  MoveC 3760 to (-84.5, 214.85, -40) mm, rotated rx 180 ry 0 rz 0.01 deg; joints [38.909, -46.829, 108.857, -137.77, 69.186, 163.004] to (-86.38, 214.39, -40) mm, rotated rx 180 ry 0 rz 0.01 deg; joints [38.847, -46.78, 108.752, -137.818, 69.125, 162.986]
  MoveC 3761 to (-98.15, 202.83, -40) mm, rotated rx 180 ry 0 rz 0.01 deg; joints [38.199, -46.687, 108.571, -138.455, 68.856, 163.166] to (-111.4, 193.01, -40) mm, rotated rx -180 ry 0 rz 0.01 deg; joints [37.571, -46.495, 108.172, -139.042, 68.504, 163.259]
  MoveC 3762 to (-125.84, 185.04, -40) mm, rotated rx -180 ry 0 rz 0.01 deg; joints [36.977, -46.211, 107.571, -139.567, 68.079, 163.268] to (-141.16, 178.95, -40) mm, rotated rx -180 ry 0 rz 0.01 deg; joints [36.427, -45.844, 106.785, -140.021, 67.589, 163.195]
  MoveC 3763 to (-159.21, 174.61, -40) mm, rotated rx 180 ry 0 rz 0.01 deg; joints [35.877, -45.331, 105.687, -140.431, 66.966, 163.013] to (-177.73, 173.15, -40) mm, rotated rx 180 ry 0 rz 0.01 deg; joints [35.415, -44.722, 104.377, -140.715, 66.278, 162.723]
  MoveL 3764 to (-214.9, 173.15, -40) mm, rotated rx 180 ry 0 rz 0.01 deg; joints [34.605, -43.391, 101.519, -141.119, 64.829, 162.022]
  MoveC 3765 to (-246.16, 177.17, -40) mm, rotated rx 180 ry 0 rz 0.01 deg; joints [34.072, -42.131, 98.82, -141.24, 63.528, 161.269] to (-275.4, 188.95, -40) mm, rotated rx 180 ry 0 rz 0.01 deg; joints [33.832, -40.711, 95.78, -140.971, 62.183, 160.244]
  MoveC 3766 to (-277.77, 191.44, -40) mm, rotated rx -180 ry 0 rz 0.01 deg; joints [33.859, -40.555, 95.444, -140.883, 62.053, 160.102] to (-278.34, 194.83, -40) mm, rotated rx 180 ry 0 rz 0.01 deg; joints [33.949, -40.446, 95.207, -140.745, 61.987, 159.965]
  MoveC 3767 to (-278.82, 198.21, -40) mm, rotated rx 180 ry 0 rz 0.01 deg; joints [34.04, -40.34, 94.977, -140.606, 61.924, 159.83] to (-281, 200.83, -40) mm, rotated rx 180 ry 0 rz 0.01 deg; joints [34.075, -40.185, 94.646, -140.51, 61.8, 159.685]
  MoveC 3768 to (-299.48, 216.47, -40) mm, rotated rx 180 ry 0 rz 0.01 deg; joints [34.167, -39.034, 92.185, -139.955, 60.828, 158.683] to (-314.43, 235.5, -40) mm, rotated rx 180 ry 0 rz 0.01 deg; joints [34.423, -37.901, 89.767, -139.21, 59.951, 157.588]
  MoveC 3769 to (-316.14, 236.14, -40) mm, rotated rx -180 ry 0 rz 0.01 deg; joints [34.408, -37.812, 89.579, -139.189, 59.87, 157.521] to (-317.24, 234.68, -40) mm, rotated rx -180 ry 0 rz 0.01 deg; joints [34.344, -37.807, 89.57, -139.255, 59.841, 157.552]
  MoveL 3770 to (-317.23, 140.25, -40) mm, rotated rx -180 ry 0 rz 0.01 deg; joints [31.537, -40.248, 94.881, -143.267, 61.027, 161.125]
  MoveC 3771 to (-316.14, 136.25, -40) mm, rotated rx 180 ry 0 rz 0.01 deg; joints [31.435, -40.388, 95.185, -143.43, 61.123, 161.29] to (-313.16, 133.37, -40) mm, rotated rx -180 ry 0 rz 0.01 deg; joints [31.402, -40.577, 95.59, -143.536, 61.286, 161.455]
  MoveC 3772 to (-302.92, 127.1, -40) mm, rotated rx 180 ry 0 rz 0.01 deg; joints [31.401, -41.135, 96.786, -143.742, 61.799, 161.885] to (-293.34, 119.87, -40) mm, rotated rx 180 ry 0 rz 0.01 deg; joints [31.358, -41.682, 97.963, -143.985, 62.294, 162.328]
  MoveC 3773 to (-284.52, 111.72, -40) mm, rotated rx -180 ry 0 rz 0.01 deg; joints [31.27, -42.213, 99.11, -144.266, 62.764, 162.779] to (-276.59, 102.69, -40) mm, rotated rx 180 ry 0 rz 0.01 deg; joints [31.136, -42.723, 100.215, -144.586, 63.206, 163.234]
  MoveC 3774 to (-269.25, 92.45, -40) mm, rotated rx 180 ry 0 rz 0.01 deg; joints [30.95, -43.231, 101.321, -144.957, 63.637, 163.71] to (-262.89, 81.57, -40) mm, rotated rx -180 ry 0 rz 0.01 deg; joints [30.72, -43.709, 102.366, -145.36, 64.034, 164.181]
  MoveC 3775 to (-256.94, 70.47, -40) mm, rotated rx -180 ry 0 rz 0.01 deg; joints [30.473, -44.17, 103.376, -145.773, 64.415, 164.643] to (-250.77, 59.49, -40) mm, rotated rx -180 ry 0 rz 0.01 deg; joints [30.23, -44.63, 104.388, -146.177, 64.803, 165.098]
  MoveC 3776 to (-247.69, 56.41, -40) mm, rotated rx -180 ry 0 rz 0.01 deg; joints [30.187, -44.808, 104.778, -146.277, 64.967, 165.248] to (-243.47, 55.28, -40) mm, rotated rx -180 ry 0 rz 0.01 deg; joints [30.231, -44.987, 105.167, -146.285, 65.154, 165.356]
  MoveL 3777 to (-150.05, 55.28, -40) mm, rotated rx 180 ry 0 rz 0.01 deg; joints [32.15, -48.283, 112.334, -145.198, 68.859, 166.917]
  MoveC 3778 to (-145.86, 56.4, -40) mm, rotated rx -180 ry 0 rz 0.01 deg; joints [32.28, -48.401, 112.591, -145.094, 69.006, 166.953] to (-142.79, 59.47, -40) mm, rotated rx 180 ry 0 rz 0.01 deg; joints [32.453, -48.442, 112.674, -144.924, 69.084, 166.913]
  MoveL 3779 to (-126.05, 89.53, -40) mm, rotated rx -180 ry 0 rz 0.01 deg; joints [33.855, -48.375, 112.466, -143.442, 69.327, 166.294]
  MoveC 3780 to (-117.05, 102.8, -40) mm, rotated rx 180 ry 0 rz 0.01 deg; joints [34.51, -48.386, 112.466, -142.765, 69.488, 166.042] to (-106.26, 114.65, -40) mm, rotated rx -180 ry 0 rz 0.01 deg; joints [35.159, -48.481, 112.649, -142.117, 69.732, 165.86]
  MoveC 3781 to (-93.93, 124.89, -40) mm, rotated rx 180 ry 0 rz 0.01 deg; joints [35.794, -48.653, 113.006, -141.508, 70.048, 165.751] to (-80.35, 133.4, -40) mm, rotated rx -180 ry 0 rz 0.01 deg; joints [36.405, -48.896, 113.525, -140.945, 70.427, 165.716]
  MoveC 3782 to (-77.37, 136.23, -40) mm, rotated rx 180 ry 0 rz 0.01 deg; joints [36.572, -48.927, 113.586, -140.781, 70.496, 165.678] to (-76.28, 140.19, -40) mm, rotated rx -180 ry 0 rz 0.01 deg; joints [36.73, -48.872, 113.457, -140.604, 70.482, 165.573]
  MoveL 3783 to (-76.28, 234.68, -40) mm, rotated rx 180 ry 0 rz 0.01 deg; joints [39.722, -46.589, 108.302, -136.865, 69.215, 162.474]
  MoveC 3784 to (-77.38, 236.14, -40) mm, rotated rx -180 ry 0 rz 0.01 deg; joints [39.739, -46.517, 108.143, -136.825, 69.157, 162.404] to (-79.08, 235.49, -40) mm, rotated rx -180 ry 0 rz 0.01 deg; joints [39.676, -46.479, 108.061, -136.877, 69.105, 162.395]
  MoveC 3785 to (-106.86, 204.97, -40) mm, rotated rx 180 ry 0 rz 0.01 deg; joints [38.053, -46.35, 107.836, -138.5, 68.512, 162.939] to (-143.36, 185.73, -40) mm, rotated rx -180 ry 0 rz 0.01 deg; joints [36.588, -45.605, 106.257, -139.779, 67.418, 162.929]
  MoveC 3786 to (-160.92, 181.53, -40) mm, rotated rx -180 ry 0 rz 0.01 deg; joints [36.055, -45.105, 105.187, -140.173, 66.811, 162.749] to (-178.91, 180.18, -40) mm, rotated rx 180 ry 0 rz 0.01 deg; joints [35.608, -44.51, 103.908, -140.444, 66.141, 162.462]
  MoveL 3787 to (-214.9, 180.27, -40) mm, rotated rx 180 ry 0 rz 0.01 deg; joints [34.825, -43.217, 101.133, -140.827, 64.738, 161.775]
  MoveC 3788 to (-244.28, 184.04, -40) mm, rotated rx -180 ry 0 rz 0.01 deg; joints [34.32, -42.031, 98.596, -140.941, 63.517, 161.063] to (-271.76, 195.1, -40) mm, rotated rx -180 ry 0 rz 0.01 deg; joints [34.09, -40.696, 95.739, -140.69, 62.255, 160.095]
  MoveC 3789 to (-276.45, 197.86, -40) mm, rotated rx -180 ry 0 rz 0.01 deg; joints [34.078, -40.442, 95.195, -140.606, 62.027, 159.894] to (-281, 200.83, -40) mm, rotated rx 180 ry 0 rz 0.01 deg; joints [34.075, -40.185, 94.646, -140.51, 61.8, 159.685]
  MoveC 3790 to (-282.99, 203.32, -40) mm, rotated rx 180 ry 0 rz 0.01 deg; joints [34.109, -40.042, 94.339, -140.418, 61.686, 159.549] to (-283.24, 206.49, -40) mm, rotated rx -180 ry 0 rz 0.01 deg; joints [34.198, -39.949, 94.137, -140.287, 61.635, 159.425]
  MoveC 3791 to (-283.44, 209.65, -40) mm, rotated rx 180 ry 0 rz 0.01 deg; joints [34.287, -39.859, 93.94, -140.156, 61.587, 159.301] to (-285.27, 212.23, -40) mm, rotated rx 180 ry 0 rz 0.01 deg; joints [34.327, -39.718, 93.638, -140.058, 61.478, 159.164]
  MoveC 3792 to (-293.65, 219.64, -40) mm, rotated rx -180 ry 0 rz 0.01 deg; joints [34.376, -39.185, 92.499, -139.792, 61.034, 158.693] to (-301.3, 227.8, -40) mm, rotated rx -180 ry 0 rz 0.01 deg; joints [34.461, -38.654, 91.365, -139.485, 60.607, 158.202]
  MoveC 3793 to (-306.53, 234.56, -40) mm, rotated rx 180 ry 0 rz 0.01 deg; joints [34.553, -38.254, 90.512, -139.22, 60.3, 157.813] to (-311.05, 241.82, -40) mm, rotated rx -180 ry 0 rz 0.01 deg; joints [34.672, -37.866, 89.683, -138.929, 60.015, 157.416]
  MoveC 3794 to (-314.94, 249.42, -40) mm, rotated rx -180 ry 0 rz 0.01 deg; joints [34.812, -37.489, 88.879, -138.618, 59.751, 157.015] to (-318.34, 257.27, -40) mm, rotated rx 180 ry 0 rz 0.01 deg; joints [34.968, -37.123, 88.098, -138.292, 59.505, 156.611]
  MoveC 3795 to (-321.51, 259.02, -40) mm, rotated rx 180 ry 0 rz 0.01 deg; joints [34.955, -36.939, 87.708, -138.225, 59.346, 156.46] to (-323.82, 256.23, -40) mm, rotated rx -180 ry 0 rz 0.01 deg; joints [34.83, -36.921, 87.676, -138.351, 59.282, 156.516]
  MoveL 3796 to (-323.81, 135.87, -40) mm, rotated rx 180 ry 0 rz 0.01 deg; joints [31.279, -40.086, 94.544, -143.485, 60.797, 161.143]
  MoveC 3797 to (-322.72, 132.05, -40) mm, rotated rx -180 ry 0 rz 0.01 deg; joints [31.182, -40.222, 94.838, -143.642, 60.892, 161.302] to (-319.77, 129.39, -40) mm, rotated rx -180 ry 0 rz 0.01 deg; joints [31.155, -40.405, 95.231, -143.74, 61.051, 161.459]
  MoveC 3798 to (-299.02, 116.16, -40) mm, rotated rx -180 ry 0 rz 0.01 deg; joints [31.134, -41.544, 97.675, -144.179, 62.099, 162.343] to (-281.76, 98.61, -40) mm, rotated rx 180 ry 0 rz 0.01 deg; joints [30.907, -42.615, 99.991, -144.796, 63.041, 163.272]
  MoveC 3799 to (-273.96, 87.77, -40) mm, rotated rx 180 ry 0 rz 0.01 deg; joints [30.708, -43.154, 101.164, -145.191, 63.499, 163.776] to (-267.18, 76.25, -40) mm, rotated rx -180 ry 0 rz 0.01 deg; joints [30.465, -43.661, 102.272, -145.619, 63.921, 164.274]
  MoveL 3800 to (-254.5, 52.76, -40) mm, rotated rx 180 ry 0 rz 0.01 deg; joints [29.935, -44.63, 104.401, -146.494, 64.732, 165.243]
  MoveC 3801 to (-251.61, 49.79, -40) mm, rotated rx 180 ry 0 rz 0.01 deg; joints [29.891, -44.798, 104.77, -146.592, 64.887, 165.385] to (-247.62, 48.7, -40) mm, rotated rx -180 ry 0 rz 0.01 deg; joints [29.932, -44.969, 105.14, -146.6, 65.064, 165.488]
  MoveL 3802 to (-145.88, 48.7, -40) mm, rotated rx 180 ry 0 rz 0.01 deg; joints [32.013, -48.555, 112.946, -145.415, 69.104, 167.177]
  MoveC 3803 to (-141.9, 49.79, -40) mm, rotated rx 180 ry 0 rz 0.01 deg; joints [32.137, -48.667, 113.189, -145.314, 69.243, 167.209] to (-139.04, 52.76, -40) mm, rotated rx -180 ry 0 rz 0.01 deg; joints [32.303, -48.703, 113.262, -145.15, 69.314, 167.169]
  MoveL 3804 to (-119.94, 86.41, -40) mm, rotated rx 180 ry 0 rz 0.01 deg; joints [33.889, -48.642, 113.058, -143.48, 69.597, 166.488]
  MoveC 3805 to (-108.73, 102.26, -40) mm, rotated rx 180 ry 0 rz 0.01 deg; joints [34.685, -48.67, 113.089, -142.66, 69.805, 166.197] to (-95.08, 116.07, -40) mm, rotated rx 180 ry 0 rz 0.01 deg; joints [35.472, -48.811, 113.37, -141.885, 70.124, 166.003]
  MoveC 3806 to (-90.13, 119.96, -40) mm, rotated rx -180 ry 0 rz 0.01 deg; joints [35.72, -48.884, 113.523, -141.647, 70.253, 165.967] to (-84.87, 123.41, -40) mm, rotated rx 180 ry 0 rz 0.01 deg; joints [35.963, -48.975, 113.718, -141.422, 70.398, 165.949]
  MoveC 3807 to (-79.39, 126.51, -40) mm, rotated rx -180 ry 0 rz 0.01 deg; joints [36.199, -49.08, 113.943, -141.207, 70.554, 165.945] to (-73.78, 129.35, -40) mm, rotated rx 180 ry 0 rz 0.01 deg; joints [36.432, -49.194, 114.189, -140.999, 70.719, 165.951]
  MoveC 3808 to (-70.8, 132, -40) mm, rotated rx -180 ry 0 rz 0.01 deg; joints [36.593, -49.229, 114.259, -140.842, 70.79, 165.92] to (-69.7, 135.82, -40) mm, rotated rx 180 ry 0 rz 0.01 deg; joints [36.747, -49.178, 114.139, -140.669, 70.777, 165.82]
  MoveL 3809 to (-69.7, 256.21, -40) mm, rotated rx -180 ry 0 rz 0.01 deg; joints [40.537, -46.238, 107.505, -135.924, 69.16, 161.843]
  MoveC 3810 to (-72.01, 259, -40) mm, rotated rx -180 ry 0 rz 0.01 deg; joints [40.562, -46.091, 107.182, -135.853, 69.042, 161.703] to (-75.18, 257.25, -40) mm, rotated rx 180 ry 0 rz 0.01 deg; joints [40.429, -46.036, 107.066, -135.97, 68.954, 161.707]
  MoveC 3811 to (-85.01, 238.11, -40) mm, rotated rx -180 ry 0 rz 0.01 deg; joints [39.607, -46.221, 107.498, -136.867, 68.859, 162.198] to (-98.4, 221.27, -40) mm, rotated rx 180 ry 0 rz 0.01 deg; joints [38.762, -46.218, 107.52, -137.731, 68.602, 162.536]
  MoveC 3812 to (-114.74, 207.28, -40) mm, rotated rx 180 ry 0 rz 0.01 deg; joints [37.934, -46.033, 107.145, -138.523, 68.194, 162.718] to (-133.35, 196.51, -40) mm, rotated rx -180 ry 0 rz 0.01 deg; joints [37.158, -45.679, 106.398, -139.212, 67.65, 162.746]
  MoveC 3813 to (-152.99, 189.8, -40) mm, rotated rx 180 ry 0 rz 0.01 deg; joints [36.493, -45.176, 105.325, -139.74, 67.003, 162.615] to (-173.6, 187.26, -40) mm, rotated rx -180 ry 0 rz 0.01 deg; joints [35.946, -44.524, 103.925, -140.095, 66.254, 162.32]
  MoveL 3814 to (-214.9, 186.85, -40) mm, rotated rx -180 ry 0 rz 0.01 deg; joints [35.027, -43.054, 100.774, -140.558, 64.654, 161.546]
  MoveC 3815 to (-239.37, 189.64, -40) mm, rotated rx 180 ry 0 rz 0.01 deg; joints [34.593, -42.076, 98.682, -140.668, 63.644, 160.962] to (-262.59, 197.85, -40) mm, rotated rx 180 ry 0 rz 0.01 deg; joints [34.36, -40.982, 96.341, -140.512, 62.598, 160.188]
  MoveC 3816 to (-274.33, 204.41, -40) mm, rotated rx 180 ry 0 rz 0.01 deg; joints [34.316, -40.356, 95.001, -140.319, 62.032, 159.696] to (-285.27, 212.23, -40) mm, rotated rx 180 ry 0 rz 0.01 deg; joints [34.327, -39.718, 93.638, -140.058, 61.478, 159.164]
  MoveC 3817 to (-287.81, 216, -40) mm, rotated rx -180 ry 0 rz 0.01 deg; joints [34.386, -39.517, 93.206, -139.914, 61.325, 158.964] to (-287.78, 220.54, -40) mm, rotated rx 180 ry 0 rz 0.01 deg; joints [34.52, -39.397, 92.945, -139.724, 61.268, 158.791]
  MoveC 3818 to (-287.6, 225.04, -40) mm, rotated rx 180 ry 0 rz 0.01 deg; joints [34.656, -39.283, 92.697, -139.534, 61.218, 158.622] to (-289.76, 229, -40) mm, rotated rx 180 ry 0 rz 0.01 deg; joints [34.727, -39.089, 92.282, -139.379, 61.078, 158.421]
  MoveC 3819 to (-292.01, 231.41, -40) mm, rotated rx -180 ry 0 rz 0.01 deg; joints [34.752, -38.933, 91.949, -139.289, 60.953, 158.276] to (-294.19, 233.88, -40) mm, rotated rx 180 ry 0 rz 0.01 deg; joints [34.78, -38.777, 91.616, -139.195, 60.83, 158.129]
  MoveC 3820 to (-299.55, 240.88, -40) mm, rotated rx 180 ry 0 rz 0.01 deg; joints [34.875, -38.366, 90.738, -138.924, 60.515, 157.728] to (-304.11, 248.43, -40) mm, rotated rx 180 ry 0 rz 0.01 deg; joints [35, -37.967, 89.887, -138.623, 60.225, 157.319]
  MoveC 3821 to (-307.93, 256.38, -40) mm, rotated rx 180 ry 0 rz 0.01 deg; joints [35.15, -37.584, 89.069, -138.298, 59.961, 156.905] to (-311.05, 264.62, -40) mm, rotated rx 180 ry 0 rz 0.01 deg; joints [35.321, -37.218, 88.285, -137.957, 59.722, 156.491]
  MoveC 3822 to (-313.15, 267.5, -40) mm, rotated rx -180 ry 0 rz 0.01 deg; joints [35.36, -37.046, 87.92, -137.84, 59.595, 156.32] to (-316.54, 268.59, -40) mm, rotated rx 180 ry 0 rz 0.01 deg; joints [35.323, -36.871, 87.552, -137.802, 59.436, 156.189]
  MoveL 3823 to (-329.33, 268.59, -40) mm, rotated rx 180 ry 0 rz 0.01 deg; joints [35.07, -36.326, 86.408, -137.829, 58.884, 155.86]
  MoveC 3824 to (-332.05, 267.47, -40) mm, rotated rx 180 ry 0 rz 0.01 deg; joints [34.985, -36.242, 86.234, -137.882, 58.78, 155.837] to (-333.18, 264.74, -40) mm, rotated rx -180 ry 0 rz 0.01 deg; joints [34.886, -36.274, 86.304, -138.002, 58.766, 155.922]
  MoveL 3825 to (-333.17, 129.66, -40) mm, rotated rx 180 ry 0 rz 0.01 deg; joints [30.915, -39.85, 94.055, -143.793, 60.468, 161.167]
  MoveC 3826 to (-332.04, 125.85, -40) mm, rotated rx 180 ry 0 rz 0.01 deg; joints [30.819, -39.987, 94.352, -143.95, 60.564, 161.327] to (-329, 123.29, -40) mm, rotated rx -180 ry 0 rz 0.01 deg; joints [30.796, -40.172, 94.749, -144.045, 60.727, 161.483]
  MoveC 3827 to (-321.93, 119.98, -40) mm, rotated rx 180 ry 0 rz 0.01 deg; joints [30.824, -40.538, 95.531, -144.15, 61.074, 161.747] to (-315.03, 116.31, -40) mm, rotated rx 180 ry 0 rz 0.01 deg; joints [30.838, -40.902, 96.309, -144.269, 61.415, 162.016]
  MoveC 3828 to (-308.46, 112.08, -40) mm, rotated rx 180 ry 0 rz 0.01 deg; joints [30.828, -41.263, 97.084, -144.409, 61.748, 162.295] to (-302.39, 107.15, -40) mm, rotated rx -180 ry 0 rz 0.01 deg; joints [30.787, -41.616, 97.845, -144.58, 62.066, 162.585]
  MoveC 3829 to (-296.35, 101.27, -40) mm, rotated rx 180 ry 0 rz 0.01 deg; joints [30.715, -41.987, 98.647, -144.788, 62.394, 162.903] to (-290.71, 95, -40) mm, rotated rx 180 ry 0 rz 0.01 deg; joints [30.622, -42.348, 99.427, -145.013, 62.709, 163.222]
  MoveC 3830 to (-285.57, 88.3, -40) mm, rotated rx -180 ry 0 rz 0.01 deg; joints [30.505, -42.695, 100.182, -145.258, 63.007, 163.542] to (-281.04, 81.19, -40) mm, rotated rx -180 ry 0 rz 0.01 deg; joints [30.361, -43.025, 100.901, -145.523, 63.283, 163.86]
  MoveL 3831 to (-263.18, 49.54, -40) mm, rotated rx 180 ry 0 rz 0.01 deg; joints [29.663, -44.371, 103.849, -146.707, 64.411, 165.192]
  MoveC 3832 to (-262.37, 48.04, -40) mm, rotated rx 180 ry 0 rz 0.01 deg; joints [29.628, -44.432, 103.984, -146.763, 64.463, 165.253] to (-261.64, 46.49, -40) mm, rotated rx -180 ry 0 rz 0.01 deg; joints [29.59, -44.491, 104.114, -146.821, 64.512, 165.314]
  MoveC 3833 to (-260.94, 44.92, -40) mm, rotated rx -180 ry 0 rz 0.01 deg; joints [29.551, -44.549, 104.242, -146.881, 64.56, 165.374] to (-260.23, 43.36, -40) mm, rotated rx -180 ry 0 rz 0.01 deg; joints [29.513, -44.608, 104.37, -146.94, 64.608, 165.435]
  MoveC 3834 to (-257.69, 40.43, -40) mm, rotated rx 180 ry 0 rz 0.01 deg; joints [29.463, -44.762, 104.709, -147.041, 64.749, 165.569] to (-253.96, 39.34, -40) mm, rotated rx 180 ry 0 rz 0.01 deg; joints [29.497, -44.923, 105.059, -147.053, 64.917, 165.666]
  MoveL 3835 to (-139.55, 39.34, -40) mm, rotated rx -180 ry 0 rz 0.01 deg; joints [31.824, -48.953, 113.84, -145.717, 69.468, 167.549]
  MoveC 3836 to (-135.8, 40.44, -40) mm, rotated rx 180 ry 0 rz 0.01 deg; joints [31.944, -49.056, 114.065, -145.618, 69.597, 167.577] to (-133.25, 43.4, -40) mm, rotated rx -180 ry 0 rz 0.01 deg; joints [32.103, -49.082, 114.116, -145.458, 69.656, 167.533]
  MoveC 3837 to (-132.51, 45.06, -40) mm, rotated rx 180 ry 0 rz 0.01 deg; joints [32.178, -49.073, 114.095, -145.378, 69.663, 167.497] to (-131.77, 46.73, -40) mm, rotated rx -180 ry 0 rz 0.01 deg; joints [32.253, -49.065, 114.072, -145.298, 69.67, 167.461]
  MoveC 3838 to (-130.99, 48.39, -40) mm, rotated rx -180 ry 0 rz 0.01 deg; joints [32.328, -49.058, 114.052, -145.217, 69.678, 167.426] to (-130.12, 49.99, -40) mm, rotated rx 180 ry 0 rz 0.01 deg; joints [32.403, -49.054, 114.042, -145.138, 69.69, 167.393]
  MoveL 3839 to (-109.71, 84.93, -40) mm, rotated rx -180 ry 0 rz 0.01 deg; joints [34.074, -49.007, 113.865, -143.386, 69.999, 166.701]
  MoveC 3840 to (-97.46, 101.2, -40) mm, rotated rx 180 ry 0 rz 0.01 deg; joints [34.914, -49.057, 113.943, -142.528, 70.235, 166.416] to (-81.91, 114.34, -40) mm, rotated rx 180 ry 0 rz 0.01 deg; joints [35.73, -49.269, 114.383, -141.742, 70.627, 166.275]
  MoveC 3841 to (-77.72, 116.92, -40) mm, rotated rx 180 ry 0 rz 0.01 deg; joints [35.919, -49.345, 114.545, -141.568, 70.744, 166.266] to (-73.36, 119.19, -40) mm, rotated rx 180 ry 0 rz 0.01 deg; joints [36.102, -49.432, 114.734, -141.403, 70.871, 166.27]
  MoveC 3842 to (-68.92, 121.27, -40) mm, rotated rx 180 ry 0 rz 0.01 deg; joints [36.281, -49.526, 114.937, -141.243, 71.003, 166.28] to (-64.45, 123.31, -40) mm, rotated rx -180 ry 0 rz 0.01 deg; joints [36.46, -49.621, 115.142, -141.084, 71.135, 166.292]
  MoveC 3843 to (-61.45, 125.88, -40) mm, rotated rx 180 ry 0 rz 0.01 deg; joints [36.621, -49.657, 115.217, -140.929, 71.207, 166.263] to (-60.34, 129.67, -40) mm, rotated rx 180 ry 0 rz 0.01 deg; joints [36.775, -49.608, 115.1, -140.757, 71.196, 166.166]
  MoveL 3844 to (-60.34, 264.75, -40) mm, rotated rx 180 ry 0 rz 0.01 deg; joints [41.031, -46.308, 107.643, -135.444, 69.374, 161.712]
  MoveC 3845 to (-61.47, 267.47, -40) mm, rotated rx 180 ry 0 rz 0.01 deg; joints [41.083, -46.2, 107.404, -135.358, 69.299, 161.595] to (-64.19, 268.6, -40) mm, rotated rx 180 ry 0 rz 0.01 deg; joints [41.046, -46.083, 107.151, -135.358, 69.189, 161.506]
  MoveL 3846 to (-76.97, 268.6, -40) mm, rotated rx -180 ry 0 rz 0.01 deg; joints [40.72, -45.676, 106.271, -135.56, 68.74, 161.272]
  MoveC 3847 to (-80.36, 267.5, -40) mm, rotated rx 180 ry 0 rz 0.01 deg; joints [40.601, -45.597, 106.101, -135.654, 68.635, 161.249] to (-82.46, 264.63, -40) mm, rotated rx 180 ry 0 rz 0.01 deg; joints [40.463, -45.606, 106.125, -135.797, 68.598, 161.312]
  MoveC 3848 to (-91.11, 245.71, -40) mm, rotated rx 180 ry 0 rz 0.01 deg; joints [39.683, -45.826, 106.632, -136.664, 68.541, 161.822] to (-103.68, 229.13, -40) mm, rotated rx -180 ry 0 rz 0.01 deg; joints [38.872, -45.845, 106.701, -137.5, 68.308, 162.17]
  MoveC 3849 to (-119.33, 215.47, -40) mm, rotated rx -180 ry 0 rz 0.01 deg; joints [38.076, -45.675, 106.357, -138.264, 67.919, 162.355] to (-137.28, 205.01, -40) mm, rotated rx -180 ry 0 rz 0.01 deg; joints [37.329, -45.335, 105.642, -138.926, 67.393, 162.385]
  MoveC 3850 to (-155.98, 198.67, -40) mm, rotated rx 180 ry 0 rz 0.01 deg; joints [36.699, -44.854, 104.616, -139.421, 66.775, 162.256] to (-175.61, 196.4, -40) mm, rotated rx 180 ry 0 rz 0.01 deg; joints [36.183, -44.227, 103.271, -139.749, 66.059, 161.967]
  MoveL 3851 to (-214.9, 196.21, -40) mm, rotated rx -180 ry 0 rz 0.01 deg; joints [35.313, -42.82, 100.258, -140.175, 64.535, 161.216]
  MoveC 3852 to (-237.36, 198.78, -40) mm, rotated rx 180 ry 0 rz 0.01 deg; joints [34.912, -41.921, 98.335, -140.275, 63.608, 160.675] to (-258.67, 206.35, -40) mm, rotated rx -180 ry 0 rz 0.01 deg; joints [34.695, -40.915, 96.184, -140.13, 62.65, 159.958]
  MoveC 3853 to (-275.2, 216.32, -40) mm, rotated rx -180 ry 0 rz 0.01 deg; joints [34.651, -40.009, 94.247, -139.827, 61.844, 159.231] to (-289.76, 229, -40) mm, rotated rx -180 ry 0 rz 0.01 deg; joints [34.727, -39.089, 92.282, -139.379, 61.078, 158.421]
  MoveC 3854 to (-291.84, 233.17, -40) mm, rotated rx 180 ry 0 rz 0.01 deg; joints [34.807, -38.891, 91.858, -139.214, 60.937, 158.211] to (-291.18, 237.79, -40) mm, rotated rx -180 ry 0 rz 0.01 deg; joints [34.954, -38.792, 91.641, -139.016, 60.906, 158.045]
  MoveC 3855 to (-290.33, 242.32, -40) mm, rotated rx -180 ry 0 rz 0.01 deg; joints [35.102, -38.701, 91.443, -138.821, 60.884, 157.887] to (-291.84, 246.68, -40) mm, rotated rx 180 ry 0 rz 0.01 deg; joints [35.197, -38.519, 91.052, -138.645, 60.765, 157.68]
  MoveC 3856 to (-299.09, 259.76, -40) mm, rotated rx 180 ry 0 rz 0.01 deg; joints [35.424, -37.854, 89.63, -138.123, 60.292, 156.984] to (-303.92, 273.92, -40) mm, rotated rx 180 ry 0 rz 0.01 deg; joints [35.726, -37.245, 88.329, -137.538, 59.906, 156.286]
  MoveC 3857 to (-305.79, 276.83, -40) mm, rotated rx -180 ry 0 rz 0.01 deg; joints [35.77, -37.082, 87.981, -137.42, 59.788, 156.118] to (-309.07, 277.96, -40) mm, rotated rx 180 ry 0 rz 0.01 deg; joints [35.736, -36.911, 87.622, -137.381, 59.634, 155.989]
  MoveL 3858 to (-338.69, 277.96, -40) mm, rotated rx 180 ry 0 rz 0.01 deg; joints [35.148, -35.643, 84.962, -137.433, 58.354, 155.215]
  MoveC 3859 to (-341.41, 276.83, -40) mm, rotated rx -180 ry 0 rz 0.01 deg; joints [35.063, -35.557, 84.785, -137.484, 58.249, 155.19] to (-342.54, 274.1, -40) mm, rotated rx 180 ry 0 rz 0.01 deg; joints [34.965, -35.589, 84.856, -137.604, 58.235, 155.276]
  MoveL 3860 to (-342.54, 123.03, -40) mm, rotated rx 180 ry 0 rz 0.01 deg; joints [30.54, -39.62, 93.58, -144.116, 60.14, 161.205]
  MoveC 3861 to (-341.45, 119.5, -40) mm, rotated rx 180 ry 0 rz 0.01 deg; joints [30.451, -39.749, 93.858, -144.262, 60.231, 161.355] to (-338.56, 117.19, -40) mm, rotated rx 180 ry 0 rz 0.01 deg; joints [30.432, -39.922, 94.23, -144.348, 60.385, 161.498]
  MoveC 3862 to (-329.9, 113.43, -40) mm, rotated rx 180 ry 0 rz 0.01 deg; joints [30.474, -40.366, 95.176, -144.469, 60.808, 161.812] to (-321.53, 109.07, -40) mm, rotated rx -180 ry 0 rz 0.01 deg; joints [30.491, -40.807, 96.12, -144.611, 61.224, 162.136]
  MoveC 3863 to (-313.58, 103.96, -40) mm, rotated rx -180 ry 0 rz 0.01 deg; joints [30.478, -41.243, 97.057, -144.783, 61.628, 162.472] to (-306.25, 98, -40) mm, rotated rx 180 ry 0 rz 0.01 deg; joints [30.426, -41.67, 97.975, -144.991, 62.013, 162.821]
  MoveC 3864 to (-295.37, 86.26, -40) mm, rotated rx 180 ry 0 rz 0.01 deg; joints [30.255, -42.359, 99.466, -145.414, 62.618, 163.424] to (-286.65, 72.84, -40) mm, rotated rx -180 ry 0 rz 0.01 deg; joints [29.985, -42.989, 100.838, -145.917, 63.149, 164.029]
  MoveL 3865 to (-271.16, 44.94, -40) mm, rotated rx 180 ry 0 rz 0.01 deg; joints [29.36, -44.164, 103.412, -146.969, 64.134, 165.195]
  MoveC 3866 to (-269.8, 42.33, -40) mm, rotated rx -180 ry 0 rz 0.01 deg; joints [29.298, -44.269, 103.642, -147.067, 64.223, 165.301] to (-268.65, 39.62, -40) mm, rotated rx -180 ry 0 rz 0.01 deg; joints [29.229, -44.367, 103.859, -147.172, 64.303, 165.405]
  MoveC 3867 to (-267.59, 36.86, -40) mm, rotated rx 180 ry 0 rz 0.01 deg; joints [29.157, -44.462, 104.07, -147.279, 64.38, 165.508] to (-266.49, 34.13, -40) mm, rotated rx -180 ry 0 rz 0.01 deg; joints [29.086, -44.558, 104.282, -147.385, 64.459, 165.611]
  MoveC 3868 to (-264.02, 31.11, -40) mm, rotated rx 180 ry 0 rz 0.01 deg; joints [29.031, -44.711, 104.618, -147.49, 64.598, 165.746] to (-260.29, 29.98, -40) mm, rotated rx 180 ry 0 rz 0.01 deg; joints [29.063, -44.874, 104.971, -147.505, 64.767, 165.844]
  MoveL 3869 to (-133.15, 29.98, -40) mm, rotated rx -180 ry 0 rz 0.01 deg; joints [31.633, -49.348, 114.732, -146.018, 69.835, 167.917]
  MoveC 3870 to (-129.52, 31.07, -40) mm, rotated rx 180 ry 0 rz 0.01 deg; joints [31.751, -49.447, 114.949, -145.92, 69.959, 167.943] to (-127.1, 34, -40) mm, rotated rx 180 ry 0 rz 0.01 deg; joints [31.908, -49.47, 114.993, -145.762, 70.014, 167.899]
  MoveC 3871 to (-125.92, 36.87, -40) mm, rotated rx -180 ry 0 rz 0.01 deg; joints [32.036, -49.452, 114.949, -145.624, 70.021, 167.836] to (-124.8, 39.77, -40) mm, rotated rx 180 ry 0 rz 0.01 deg; joints [32.163, -49.432, 114.898, -145.487, 70.026, 167.772]
  MoveC 3872 to (-123.59, 42.63, -40) mm, rotated rx -180 ry 0 rz 0.01 deg; joints [32.29, -49.416, 114.855, -145.349, 70.034, 167.709] to (-122.15, 45.39, -40) mm, rotated rx 180 ry 0 rz 0.01 deg; joints [32.419, -49.408, 114.833, -145.213, 70.053, 167.653]
  MoveL 3873 to (-103.09, 78.38, -40) mm, rotated rx -180 ry 0 rz 0.01 deg; joints [34.002, -49.359, 114.654, -143.554, 70.332, 167.003]
  MoveC 3874 to (-91.51, 93.98, -40) mm, rotated rx -180 ry 0 rz 0.01 deg; joints [34.81, -49.402, 114.718, -142.729, 70.551, 166.73] to (-76.7, 106.56, -40) mm, rotated rx 180 ry 0 rz 0.01 deg; joints [35.594, -49.603, 115.136, -141.972, 70.921, 166.597]
  MoveC 3875 to (-71.53, 109.71, -40) mm, rotated rx 180 ry 0 rz 0.01 deg; joints [35.827, -49.697, 115.338, -141.756, 71.066, 166.587] to (-66.12, 112.43, -40) mm, rotated rx -180 ry 0 rz 0.01 deg; joints [36.052, -49.807, 115.576, -141.554, 71.224, 166.594]
  MoveC 3876 to (-60.57, 114.85, -40) mm, rotated rx 180 ry 0 rz 0.01 deg; joints [36.271, -49.927, 115.837, -141.36, 71.39, 166.613] to (-54.97, 117.14, -40) mm, rotated rx -180 ry 0 rz 0.01 deg; joints [36.488, -50.051, 116.105, -141.168, 71.558, 166.636]
  MoveC 3877 to (-52.07, 119.47, -40) mm, rotated rx -180 ry 0 rz 0.01 deg; joints [36.64, -50.089, 116.186, -141.023, 71.63, 166.613] to (-50.97, 123.03, -40) mm, rotated rx 180 ry 0 rz 0.01 deg; joints [36.787, -50.045, 116.08, -140.86, 71.62, 166.524]
  MoveL 3878 to (-50.98, 274.11, -40) mm, rotated rx 180 ry 0 rz 0.01 deg; joints [41.551, -46.351, 107.721, -134.932, 69.575, 161.55]
  MoveC 3879 to (-52.11, 276.84, -40) mm, rotated rx -180 ry 0 rz 0.01 deg; joints [41.601, -46.242, 107.481, -134.846, 69.499, 161.432] to (-54.83, 277.96, -40) mm, rotated rx -180 ry 0 rz 0.01 deg; joints [41.564, -46.127, 107.229, -134.848, 69.39, 161.343]
  MoveL 3880 to (-84.49, 277.96, -40) mm, rotated rx -180 ry 0 rz 0.01 deg; joints [40.804, -45.181, 105.188, -135.312, 68.351, 160.797]
  MoveC 3881 to (-87.75, 276.83, -40) mm, rotated rx 180 ry 0 rz 0.01 deg; joints [40.689, -45.106, 105.028, -135.405, 68.25, 160.777] to (-89.6, 273.92, -40) mm, rotated rx 180 ry 0 rz 0.01 deg; joints [40.557, -45.125, 105.073, -135.545, 68.222, 160.847]
  MoveC 3882 to (-96.33, 255.35, -40) mm, rotated rx -180 ry 0 rz 0.01 deg; joints [39.841, -45.403, 105.702, -136.365, 68.227, 161.386] to (-107.12, 238.8, -40) mm, rotated rx -180 ry 0 rz 0.01 deg; joints [39.08, -45.482, 105.901, -137.17, 68.056, 161.77]
  MoveC 3883 to (-121.34, 225.1, -40) mm, rotated rx 180 ry 0 rz 0.01 deg; joints [38.321, -45.363, 105.668, -137.911, 67.718, 161.985] to (-138.23, 214.88, -40) mm, rotated rx 180 ry 0 rz 0.01 deg; joints [37.609, -45.055, 105.019, -138.545, 67.229, 162.027]
  MoveC 3884 to (-147.91, 210.98, -40) mm, rotated rx -180 ry 0 rz 0.01 deg; joints [37.263, -44.823, 104.528, -138.826, 66.919, 161.982] to (-157.92, 208.04, -40) mm, rotated rx 180 ry 0 rz 0.01 deg; joints [36.942, -44.553, 103.951, -139.069, 66.581, 161.897]
  MoveC 3885 to (-168.2, 206.2, -40) mm, rotated rx 180 ry 0 rz 0.01 deg; joints [36.651, -44.242, 103.286, -139.268, 66.215, 161.767] to (-178.62, 205.58, -40) mm, rotated rx -180 ry 0 rz 0.01 deg; joints [36.396, -43.891, 102.534, -139.413, 65.825, 161.59]
  MoveL 3886 to (-217.25, 205.68, -40) mm, rotated rx -180 ry 0 rz 0.01 deg; joints [35.549, -42.494, 99.545, -139.811, 64.321, 160.832]
  MoveC 3887 to (-236.55, 208.01, -40) mm, rotated rx -180 ry 0 rz 0.01 deg; joints [35.207, -41.715, 97.882, -139.888, 63.523, 160.357] to (-254.82, 214.67, -40) mm, rotated rx -180 ry 0 rz 0.01 deg; joints [35.022, -40.846, 96.025, -139.758, 62.701, 159.732]
  MoveC 3888 to (-271.56, 225.24, -40) mm, rotated rx 180 ry 0 rz 0.01 deg; joints [34.988, -39.915, 94.034, -139.433, 61.881, 158.973] to (-285.89, 238.89, -40) mm, rotated rx 180 ry 0 rz 0.01 deg; joints [35.093, -38.975, 92.025, -138.943, 61.113, 158.124]
  MoveC 3889 to (-288.98, 242.7, -40) mm, rotated rx 180 ry 0 rz 0.01 deg; joints [35.14, -38.745, 91.535, -138.799, 60.936, 157.904] to (-291.84, 246.68, -40) mm, rotated rx 180 ry 0 rz 0.01 deg; joints [35.197, -38.519, 91.052, -138.645, 60.765, 157.68]
  MoveC 3890 to (-293.12, 250.97, -40) mm, rotated rx -180 ry 0 rz 0.01 deg; joints [35.294, -38.347, 90.682, -138.47, 60.656, 157.48] to (-291.71, 255.22, -40) mm, rotated rx -180 ry 0 rz 0.01 deg; joints [35.444, -38.285, 90.545, -138.284, 60.661, 157.343]
  MoveC 3891 to (-290.12, 259.34, -40) mm, rotated rx 180 ry 0 rz 0.01 deg; joints [35.594, -38.233, 90.429, -138.103, 60.675, 157.216] to (-290.76, 263.71, -40) mm, rotated rx 180 ry 0 rz 0.01 deg; joints [35.705, -38.083, 90.106, -137.922, 60.592, 157.025]
  MoveC 3892 to (-291.59, 265.76, -40) mm, rotated rx -180 ry 0 rz 0.01 deg; joints [35.746, -37.99, 89.907, -137.839, 60.53, 156.922] to (-292.37, 267.83, -40) mm, rotated rx 180 ry 0 rz 0.01 deg; joints [35.789, -37.899, 89.712, -137.754, 60.471, 156.819]
  MoveC 3893 to (-294.26, 273.68, -40) mm, rotated rx -180 ry 0 rz 0.01 deg; joints [35.916, -37.652, 89.184, -137.514, 60.316, 156.534] to (-295.79, 279.64, -40) mm, rotated rx -180 ry 0 rz 0.01 deg; joints [36.052, -37.415, 88.677, -137.267, 60.175, 156.251]
  MoveC 3894 to (-295.98, 280.55, -40) mm, rotated rx 180 ry 0 rz 0.01 deg; joints [36.074, -37.38, 88.603, -137.229, 60.155, 156.209] to (-296.14, 281.47, -40) mm, rotated rx -180 ry 0 rz 0.01 deg; joints [36.096, -37.347, 88.531, -137.191, 60.137, 156.167]
  MoveC 3895 to (-296.3, 282.38, -40) mm, rotated rx 180 ry 0 rz 0.01 deg; joints [36.119, -37.313, 88.46, -137.153, 60.118, 156.126] to (-296.48, 283.29, -40) mm, rotated rx 180 ry 0 rz 0.01 deg; joints [36.14, -37.279, 88.386, -137.115, 60.099, 156.083]
  MoveC 3896 to (-298.29, 286.19, -40) mm, rotated rx -180 ry 0 rz 0.01 deg; joints [36.184, -37.118, 88.044, -136.998, 59.985, 155.917] to (-301.51, 287.32, -40) mm, rotated rx -180 ry 0 rz 0.01 deg; joints [36.15, -36.95, 87.69, -136.96, 59.834, 155.789]
  MoveL 3897 to (-348.05, 287.32, -40) mm, rotated rx -180 ry 0 rz 0.01 deg; joints [35.224, -34.946, 83.49, -137.025, 57.82, 154.551]
  MoveC 3898 to (-350.78, 286.19, -40) mm, rotated rx 180 ry 0 rz 0.01 deg; joints [35.14, -34.859, 83.31, -137.074, 57.714, 154.525] to (-351.9, 283.47, -40) mm, rotated rx 180 ry 0 rz 0.01 deg; joints [35.043, -34.892, 83.383, -137.193, 57.699, 154.613]
  MoveL 3899 to (-351.9, 115.53, -40) mm, rotated rx 180 ry 0 rz 0.01 deg; joints [30.141, -39.406, 93.14, -144.473, 59.819, 161.274]
  MoveC 3900 to (-350.81, 112.32, -40) mm, rotated rx 180 ry 0 rz 0.01 deg; joints [30.061, -39.527, 93.401, -144.606, 59.906, 161.412] to (-348, 110.45, -40) mm, rotated rx 180 ry 0 rz 0.01 deg; joints [30.054, -39.688, 93.745, -144.675, 60.053, 161.539]
  MoveC 3901 to (-321.73, 98.25, -40) mm, rotated rx -180 ry 0 rz 0.01 deg; joints [30.148, -41.045, 96.645, -145.071, 61.346, 162.506] to (-301.24, 77.78, -40) mm, rotated rx 180 ry 0 rz 0.01 deg; joints [29.874, -42.313, 99.384, -145.812, 62.471, 163.594]
  MoveC 3902 to (-286.18, 53.51, -40) mm, rotated rx 180 ry 0 rz 0.01 deg; joints [29.364, -43.414, 101.785, -146.728, 63.401, 164.659] to (-273.87, 27.74, -40) mm, rotated rx -180 ry 0 rz 0.01 deg; joints [28.735, -44.407, 103.969, -147.718, 64.227, 165.681]
  MoveC 3903 to (-273.57, 26.95, -40) mm, rotated rx -180 ry 0 rz 0.01 deg; joints [28.714, -44.434, 104.028, -147.748, 64.249, 165.71] to (-273.3, 26.15, -40) mm, rotated rx 180 ry 0 rz 0.01 deg; joints [28.693, -44.46, 104.086, -147.78, 64.27, 165.739]
  MoveC 3904 to (-273.05, 25.35, -40) mm, rotated rx -180 ry 0 rz 0.01 deg; joints [28.67, -44.485, 104.142, -147.812, 64.29, 165.768] to (-272.79, 24.55, -40) mm, rotated rx 180 ry 0 rz 0.01 deg; joints [28.648, -44.511, 104.199, -147.843, 64.311, 165.797]
  MoveC 3905 to (-270.66, 21.7, -40) mm, rotated rx 180 ry 0 rz 0.01 deg; joints [28.591, -44.647, 104.499, -147.946, 64.433, 165.92] to (-267.28, 20.62, -40) mm, rotated rx -180 ry 0 rz 0.01 deg; joints [28.617, -44.796, 104.822, -147.962, 64.588, 166.01]
  MoveL 3906 to (-126.31, 20.62, -40) mm, rotated rx 180 ry 0 rz 0.01 deg; joints [31.449, -49.754, 115.651, -146.312, 70.218, 168.287]
  MoveC 3907 to (-122.89, 21.7, -40) mm, rotated rx -180 ry 0 rz 0.01 deg; joints [31.563, -49.845, 115.851, -146.216, 70.334, 168.311] to (-120.72, 24.55, -40) mm, rotated rx 180 ry 0 rz 0.01 deg; joints [31.713, -49.862, 115.881, -146.064, 70.38, 168.265]
  MoveC 3908 to (-115.57, 37.15, -40) mm, rotated rx -180 ry 0 rz 0.01 deg; joints [32.276, -49.786, 115.686, -145.458, 70.41, 167.992] to (-109.29, 49.24, -40) mm, rotated rx 180 ry 0 rz 0.01 deg; joints [32.844, -49.751, 115.583, -144.858, 70.487, 167.749]
  MoveL 3909 to (-96.03, 72.18, -40) mm, rotated rx 180 ry 0 rz 0.01 deg; joints [33.952, -49.714, 115.452, -143.698, 70.676, 167.299]
  MoveC 3910 to (-86.53, 85.34, -40) mm, rotated rx -180 ry 0 rz 0.01 deg; joints [34.632, -49.744, 115.49, -143.002, 70.85, 167.068] to (-74.56, 96.31, -40) mm, rotated rx -180 ry 0 rz 0.01 deg; joints [35.296, -49.89, 115.792, -142.354, 71.138, 166.938]
  MoveC 3911 to (-60.7, 104.74, -40) mm, rotated rx -180 ry 0 rz 0.01 deg; joints [35.924, -50.143, 116.334, -141.772, 71.523, 166.914] to (-45.52, 110.45, -40) mm, rotated rx 180 ry 0 rz 0.01 deg; joints [36.499, -50.487, 117.087, -141.27, 71.986, 166.992]
  MoveC 3912 to (-42.7, 112.35, -40) mm, rotated rx 180 ry 0 rz 0.01 deg; joints [36.635, -50.532, 117.183, -141.142, 72.06, 166.982] to (-41.61, 115.57, -40) mm, rotated rx -180 ry 0 rz 0.01 deg; joints [36.772, -50.495, 117.095, -140.992, 72.054, 166.903]
  MoveL 3913 to (-41.61, 283.47, -40) mm, rotated rx -180 ry 0 rz 0.01 deg; joints [42.071, -46.389, 107.788, -134.418, 69.772, 161.385]
  MoveC 3914 to (-42.74, 286.2, -40) mm, rotated rx 180 ry 0 rz 0.01 deg; joints [42.121, -46.28, 107.547, -134.333, 69.697, 161.267] to (-45.47, 287.33, -40) mm, rotated rx -180 ry 0 rz 0.01 deg; joints [42.082, -46.165, 107.296, -134.336, 69.589, 161.177]
  MoveL 3915 to (-91.94, 287.33, -40) mm, rotated rx -180 ry 0 rz 0.01 deg; joints [40.889, -44.683, 104.1, -135.06, 67.963, 160.316]
  MoveC 3916 to (-95.17, 286.2, -40) mm, rotated rx -180 ry 0 rz 0.01 deg; joints [40.776, -44.608, 103.941, -135.15, 67.862, 160.296] to (-97, 283.32, -40) mm, rotated rx 180 ry 0 rz 0.01 deg; joints [40.647, -44.627, 103.986, -135.288, 67.835, 160.367]
  MoveL 3917 to (-99.67, 271.84, -40) mm, rotated rx 180 ry 0 rz 0.01 deg; joints [40.245, -44.852, 104.488, -135.772, 67.89, 160.733]
  MoveC 3918 to (-101.39, 266.18, -40) mm, rotated rx 180 ry 0 rz 0.01 deg; joints [40.036, -44.948, 104.704, -136.017, 67.902, 160.905] to (-103.89, 260.82, -40) mm, rotated rx 180 ry 0 rz 0.01 deg; joints [39.817, -45.009, 104.845, -136.261, 67.883, 161.051]
  MoveC 3919 to (-117.37, 242.31, -40) mm, rotated rx -180 ry 0 rz 0.01 deg; joints [38.936, -45.051, 104.966, -137.177, 67.638, 161.457] to (-134.99, 227.68, -40) mm, rotated rx -180 ry 0 rz 0.01 deg; joints [38.074, -44.838, 104.531, -137.993, 67.182, 161.642]
  MoveC 3920 to (-155.89, 218.19, -40) mm, rotated rx -180 ry 0 rz 0.01 deg; joints [37.298, -44.366, 103.531, -138.638, 66.525, 161.581] to (-178.62, 214.94, -40) mm, rotated rx -180 ry 0 rz 0.01 deg; joints [36.681, -43.653, 102.009, -139.036, 65.704, 161.261]
  MoveL 3921 to (-221.2, 215.57, -40) mm, rotated rx -180 ry 0 rz 0.01 deg; joints [35.761, -42.094, 98.676, -139.444, 64.038, 160.396]
  MoveC 3922 to (-242.39, 219.41, -40) mm, rotated rx 180 ry 0 rz 0.01 deg; joints [35.423, -41.198, 96.764, -139.467, 63.144, 159.818] to (-261.5, 229.33, -40) mm, rotated rx 180 ry 0 rz 0.01 deg; joints [35.316, -40.2, 94.63, -139.197, 62.242, 159.038]
  MoveC 3923 to (-268.93, 235.17, -40) mm, rotated rx 180 ry 0 rz 0.01 deg; joints [35.333, -39.751, 93.671, -139.002, 61.863, 158.652] to (-275.9, 241.56, -40) mm, rotated rx -180 ry 0 rz 0.01 deg; joints [35.374, -39.301, 92.71, -138.777, 61.494, 158.249]
  MoveC 3924 to (-282.14, 248.68, -40) mm, rotated rx -180 ry 0 rz 0.01 deg; joints [35.452, -38.855, 91.757, -138.513, 61.144, 157.827] to (-287.3, 256.62, -40) mm, rotated rx -180 ry 0 rz 0.01 deg; joints [35.574, -38.424, 90.836, -138.205, 60.827, 157.392]
  MoveC 3925 to (-289.12, 260.12, -40) mm, rotated rx 180 ry 0 rz 0.01 deg; joints [35.637, -38.251, 90.467, -138.066, 60.706, 157.208] to (-290.76, 263.71, -40) mm, rotated rx 180 ry 0 rz 0.01 deg; joints [35.705, -38.083, 90.106, -137.922, 60.592, 157.025]
  MoveC 3926 to (-291.22, 268.09, -40) mm, rotated rx 180 ry 0 rz 0.01 deg; joints [35.82, -37.938, 89.795, -137.738, 60.516, 156.836] to (-289.15, 271.99, -40) mm, rotated rx 180 ry 0 rz 0.01 deg; joints [35.973, -37.91, 89.73, -137.565, 60.552, 156.728]
  MoveC 3927 to (-286.92, 275.73, -40) mm, rotated rx -180 ry 0 rz 0.01 deg; joints [36.124, -37.893, 89.688, -137.398, 60.597, 156.63] to (-286.73, 280.07, -40) mm, rotated rx 180 ry 0 rz 0.01 deg; joints [36.25, -37.774, 89.432, -137.214, 60.549, 156.456]
  MoveC 3928 to (-287.89, 286.46, -40) mm, rotated rx -180 ry 0 rz 0.01 deg; joints [36.405, -37.539, 88.929, -136.949, 60.418, 156.165] to (-288.76, 292.89, -40) mm, rotated rx 180 ry 0 rz 0.01 deg; joints [36.567, -37.313, 88.444, -136.68, 60.299, 155.877]
  MoveC 3929 to (-290.15, 295.6, -40) mm, rotated rx -180 ry 0 rz 0.01 deg; joints [36.613, -37.175, 88.149, -136.571, 60.205, 155.729] to (-293, 296.68, -40) mm, rotated rx 180 ry 0 rz 0.01 deg; joints [36.585, -37.025, 87.832, -136.534, 60.072, 155.611]
  MoveL 3930 to (-357.41, 296.68, -40) mm, rotated rx -180 ry 0 rz 0.01 deg; joints [35.299, -34.236, 81.993, -136.603, 57.28, 153.87]
  MoveC 3931 to (-360.14, 295.55, -40) mm, rotated rx 180 ry 0 rz 0.01 deg; joints [35.216, -34.147, 81.81, -136.65, 57.173, 153.841] to (-361.27, 292.83, -40) mm, rotated rx -180 ry 0 rz 0.01 deg; joints [35.12, -34.181, 81.885, -136.769, 57.158, 153.931]
  MoveL 3932 to (-361.26, 107.57, -40) mm, rotated rx 180 ry 0 rz 0.01 deg; joints [29.729, -39.198, 92.714, -144.846, 59.5, 161.358]
  MoveC 3933 to (-360.16, 104.51, -40) mm, rotated rx -180 ry 0 rz 0.01 deg; joints [29.654, -39.316, 92.967, -144.974, 59.585, 161.491] to (-357.38, 102.86, -40) mm, rotated rx -180 ry 0 rz 0.01 deg; joints [29.652, -39.471, 93.299, -145.036, 59.73, 161.61]
  MoveC 3934 to (-353.91, 102.2, -40) mm, rotated rx 180 ry 0 rz 0.01 deg; joints [29.693, -39.632, 93.641, -145.051, 59.891, 161.707] to (-350.43, 101.57, -40) mm, rotated rx -180 ry 0 rz 0.01 deg; joints [29.735, -39.792, 93.98, -145.065, 60.053, 161.802]
  MoveC 3935 to (-346.99, 100.74, -40) mm, rotated rx -180 ry 0 rz 0.01 deg; joints [29.77, -39.954, 94.325, -145.087, 60.214, 161.904] to (-343.67, 99.52, -40) mm, rotated rx -180 ry 0 rz 0.01 deg; joints [29.792, -40.12, 94.678, -145.125, 60.375, 162.015]
  MoveC 3936 to (-332.37, 93.68, -40) mm, rotated rx -180 ry 0 rz 0.01 deg; joints [29.812, -40.716, 95.955, -145.321, 60.94, 162.449] to (-321.93, 86.42, -40) mm, rotated rx 180 ry 0 rz 0.01 deg; joints [29.771, -41.301, 97.212, -145.575, 61.481, 162.906]
  MoveC 3937 to (-312.75, 77.57, -40) mm, rotated rx -180 ry 0 rz 0.01 deg; joints [29.656, -41.863, 98.424, -145.896, 61.982, 163.382] to (-305.37, 67.16, -40) mm, rotated rx -180 ry 0 rz 0.01 deg; joints [29.456, -42.379, 99.545, -146.289, 62.423, 163.865]
  MoveL 3938 to (-290.63, 42.14, -40) mm, rotated rx -180 ry 0 rz 0.01 deg; joints [28.908, -43.476, 101.94, -147.242, 63.349, 164.94]
  MoveC 3939 to (-284.15, 29.09, -40) mm, rotated rx -180 ry 0 rz 0.01 deg; joints [28.593, -43.989, 103.066, -147.744, 63.779, 165.461] to (-279.86, 15.16, -40) mm, rotated rx -180 ry 0 rz 0.01 deg; joints [28.203, -44.427, 104.036, -148.299, 64.125, 165.962]
  MoveC 3940 to (-278.11, 12.35, -40) mm, rotated rx 180 ry 0 rz 0.01 deg; joints [28.14, -44.548, 104.302, -148.404, 64.231, 166.077] to (-274.98, 11.25, -40) mm, rotated rx -180 ry 0 rz 0.01 deg; joints [28.159, -44.687, 104.605, -148.424, 64.376, 166.163]
  MoveL 3941 to (-118.59, 11.25, -40) mm, rotated rx -180 ry 0 rz 0.01 deg; joints [31.282, -50.184, 116.625, -146.593, 70.635, 168.667]
  MoveC 3942 to (-115.4, 12.38, -40) mm, rotated rx 180 ry 0 rz 0.01 deg; joints [31.393, -50.267, 116.807, -146.497, 70.741, 168.685] to (-113.62, 15.27, -40) mm, rotated rx -180 ry 0 rz 0.01 deg; joints [31.536, -50.27, 116.807, -146.348, 70.771, 168.633]
  MoveC 3943 to (-112.31, 20.67, -40) mm, rotated rx 180 ry 0 rz 0.01 deg; joints [31.76, -50.21, 116.663, -146.1, 70.75, 168.505] to (-110.67, 25.98, -40) mm, rotated rx -180 ry 0 rz 0.01 deg; joints [31.987, -50.161, 116.543, -145.852, 70.742, 168.383]
  MoveC 3944 to (-108.62, 31.15, -40) mm, rotated rx -180 ry 0 rz 0.01 deg; joints [32.218, -50.128, 116.458, -145.603, 70.751, 168.271] to (-106.07, 36.1, -40) mm, rotated rx 180 ry 0 rz 0.01 deg; joints [32.452, -50.114, 116.417, -145.357, 70.782, 168.172]
  MoveL 3945 to (-84.46, 72.66, -40) mm, rotated rx 180 ry 0 rz 0.01 deg; joints [34.241, -50.073, 116.246, -143.491, 71.096, 167.472]
  MoveC 3946 to (-75.24, 82.93, -40) mm, rotated rx 180 ry 0 rz 0.01 deg; joints [34.819, -50.151, 116.398, -142.914, 71.295, 167.322] to (-64.59, 91.72, -40) mm, rotated rx -180 ry 0 rz 0.01 deg; joints [35.381, -50.299, 116.709, -142.372, 71.561, 167.237]
  MoveC 3947 to (-52.48, 98.44, -40) mm, rotated rx 180 ry 0 rz 0.01 deg; joints [35.912, -50.531, 117.211, -141.884, 71.904, 167.236] to (-39.21, 102.39, -40) mm, rotated rx 180 ry 0 rz 0.01 deg; joints [36.382, -50.853, 117.919, -141.483, 72.321, 167.335]
  MoveC 3948 to (-38.46, 102.52, -40) mm, rotated rx 180 ry 0 rz 0.01 deg; joints [36.405, -50.873, 117.963, -141.464, 72.346, 167.344] to (-37.71, 102.62, -40) mm, rotated rx 180 ry 0 rz 0.01 deg; joints [36.428, -50.894, 118.009, -141.446, 72.371, 167.353]
  MoveC 3949 to (-36.96, 102.72, -40) mm, rotated rx -180 ry 0 rz 0.01 deg; joints [36.45, -50.914, 118.054, -141.428, 72.396, 167.362] to (-36.22, 102.84, -40) mm, rotated rx -180 ry 0 rz 0.01 deg; joints [36.473, -50.934, 118.099, -141.409, 72.421, 167.371]
  MoveC 3950 to (-33.37, 104.5, -40) mm, rotated rx 180 ry 0 rz 0.01 deg; joints [36.603, -50.985, 118.208, -141.289, 72.498, 167.368] to (-32.25, 107.6, -40) mm, rotated rx -180 ry 0 rz 0.01 deg; joints [36.738, -50.952, 118.128, -141.142, 72.494, 167.294]
  MoveL 3951 to (-32.25, 292.84, -40) mm, rotated rx -180 ry 0 rz 0.01 deg; joints [42.591, -46.422, 107.844, -133.903, 69.967, 161.218]
  MoveC 3952 to (-33.38, 295.56, -40) mm, rotated rx -180 ry 0 rz 0.01 deg; joints [42.64, -46.312, 107.603, -133.82, 69.893, 161.1] to (-36.11, 296.69, -40) mm, rotated rx -180 ry 0 rz 0.01 deg; joints [42.6, -46.198, 107.352, -133.824, 69.785, 161.009]
  MoveL 3953 to (-100.55, 296.69, -40) mm, rotated rx 180 ry 0 rz 0.01 deg; joints [40.944, -44.14, 102.92, -134.82, 67.532, 159.807]
  MoveC 3954 to (-103.38, 295.6, -40) mm, rotated rx -180 ry 0 rz 0.01 deg; joints [40.842, -44.077, 102.786, -134.902, 67.445, 159.793] to (-104.75, 292.9, -40) mm, rotated rx -180 ry 0 rz 0.01 deg; joints [40.731, -44.107, 102.854, -135.026, 67.431, 159.867]
  MoveC 3955 to (-106.47, 282.43, -40) mm, rotated rx 180 ry 0 rz 0.01 deg; joints [40.386, -44.339, 103.368, -135.456, 67.506, 160.219] to (-109.43, 272.25, -40) mm, rotated rx -180 ry 0 rz 0.01 deg; joints [40.017, -44.518, 103.77, -135.893, 67.533, 160.534]
  MoveC 3956 to (-113.76, 262.56, -40) mm, rotated rx -180 ry 0 rz 0.01 deg; joints [39.626, -44.636, 104.038, -136.332, 67.503, 160.802] to (-119.5, 253.63, -40) mm, rotated rx 180 ry 0 rz 0.01 deg; joints [39.222, -44.682, 104.152, -136.761, 67.411, 161.014]
  MoveC 3957 to (-125.72, 246.48, -40) mm, rotated rx 180 ry 0 rz 0.01 deg; joints [38.86, -44.662, 104.121, -137.126, 67.277, 161.152] to (-132.85, 240.25, -40) mm, rotated rx 180 ry 0 rz 0.01 deg; joints [38.503, -44.584, 103.965, -137.467, 67.096, 161.239]
  MoveC 3958 to (-140.69, 234.94, -40) mm, rotated rx -180 ry 0 rz 0.01 deg; joints [38.158, -44.456, 103.699, -137.779, 66.876, 161.279] to (-149.05, 230.51, -40) mm, rotated rx -180 ry 0 rz 0.01 deg; joints [37.829, -44.285, 103.337, -138.061, 66.622, 161.277]
  MoveC 3959 to (-154.63, 228.32, -40) mm, rotated rx -180 ry 0 rz 0.01 deg; joints [37.633, -44.149, 103.049, -138.217, 66.441, 161.248] to (-160.42, 226.78, -40) mm, rotated rx 180 ry 0 rz 0.01 deg; joints [37.452, -43.988, 102.706, -138.349, 66.243, 161.192]
  MoveC 3960 to (-166.3, 225.67, -40) mm, rotated rx 180 ry 0 rz 0.01 deg; joints [37.284, -43.811, 102.329, -138.463, 66.035, 161.118] to (-172.22, 224.75, -40) mm, rotated rx -180 ry 0 rz 0.01 deg; joints [37.121, -43.627, 101.937, -138.569, 65.822, 161.037]
  MoveL 3961 to (-214.9, 224.3, -40) mm, rotated rx -180 ry 0 rz 0.01 deg; joints [36.158, -42.1, 98.674, -139.029, 64.175, 160.206]
  MoveC 3962 to (-235.16, 227.22, -40) mm, rotated rx -180 ry 0 rz 0.01 deg; joints [35.808, -41.266, 96.896, -139.087, 63.334, 159.681] to (-253.77, 235.75, -40) mm, rotated rx -180 ry 0 rz 0.01 deg; joints [35.665, -40.327, 94.89, -138.878, 62.475, 158.963]
  MoveC 3963 to (-269.43, 248.83, -40) mm, rotated rx 180 ry 0 rz 0.01 deg; joints [35.718, -39.357, 92.817, -138.436, 61.668, 158.112] to (-281.43, 265.35, -40) mm, rotated rx 180 ry 0 rz 0.01 deg; joints [35.943, -38.414, 90.802, -137.81, 60.96, 157.181]
  MoveC 3964 to (-284.44, 271.87, -40) mm, rotated rx 180 ry 0 rz 0.01 deg; joints [36.066, -38.106, 90.142, -137.55, 60.751, 156.847] to (-286.46, 278.76, -40) mm, rotated rx -180 ry 0 rz 0.01 deg; joints [36.219, -37.824, 89.539, -137.268, 60.578, 156.517]
  MoveC 3965 to (-286.6, 279.42, -40) mm, rotated rx 180 ry 0 rz 0.01 deg; joints [36.235, -37.799, 89.485, -137.241, 60.564, 156.487] to (-286.73, 280.07, -40) mm, rotated rx 180 ry 0 rz 0.01 deg; joints [36.25, -37.774, 89.432, -137.214, 60.549, 156.456]
  MoveC 3966 to (-286.32, 284.45, -40) mm, rotated rx -180 ry 0 rz 0.01 deg; joints [36.381, -37.663, 89.191, -137.028, 60.51, 156.287] to (-283.54, 287.85, -40) mm, rotated rx 180 ry 0 rz 0.01 deg; joints [36.534, -37.676, 89.215, -136.873, 60.582, 156.215]
  MoveC 3967 to (-280.65, 291.08, -40) mm, rotated rx -180 ry 0 rz 0.01 deg; joints [36.684, -37.699, 89.257, -136.724, 60.66, 156.152] to (-279.67, 295.3, -40) mm, rotated rx -180 ry 0 rz 0.01 deg; joints [36.822, -37.613, 89.071, -136.542, 60.646, 156.001]
  MoveC 3968 to (-279.65, 298.86, -40) mm, rotated rx 180 ry 0 rz 0.01 deg; joints [36.922, -37.508, 88.844, -136.392, 60.601, 155.854] to (-279.43, 302.41, -40) mm, rotated rx 180 ry 0 rz 0.01 deg; joints [37.025, -37.411, 88.635, -136.242, 60.564, 155.711]
  MoveC 3969 to (-280.29, 304.96, -40) mm, rotated rx 180 ry 0 rz 0.01 deg; joints [37.077, -37.299, 88.396, -136.138, 60.496, 155.583] to (-282.75, 306.05, -40) mm, rotated rx 180 ry 0 rz 0.01 deg; joints [37.056, -37.165, 88.114, -136.101, 60.379, 155.476]
  MoveL 3970 to (-366.78, 306.04, -40) mm, rotated rx -180 ry 0 rz 0.01 deg; joints [35.373, -33.511, 80.467, -136.167, 56.735, 153.168]
  MoveC 3971 to (-369.5, 304.92, -40) mm, rotated rx 180 ry 0 rz 0.01 deg; joints [35.29, -33.421, 80.282, -136.21, 56.626, 153.137] to (-370.63, 302.19, -40) mm, rotated rx -180 ry 0 rz 0.01 deg; joints [35.195, -33.456, 80.358, -136.33, 56.611, 153.228]
  MoveL 3972 to (-370.62, 98.54, -40) mm, rotated rx 180 ry 0 rz 0.01 deg; joints [29.287, -39.01, 92.331, -145.264, 59.189, 161.48]
  MoveC 3973 to (-369.54, 95.83, -40) mm, rotated rx -180 ry 0 rz 0.01 deg; joints [29.222, -39.118, 92.564, -145.377, 59.27, 161.6] to (-366.9, 94.62, -40) mm, rotated rx 180 ry 0 rz 0.01 deg; joints [29.23, -39.259, 92.863, -145.422, 59.404, 161.7]
  MoveC 3974 to (-344.51, 89.56, -40) mm, rotated rx 180 ry 0 rz 0.01 deg; joints [29.465, -40.311, 95.101, -145.555, 60.458, 162.346] to (-325.15, 77.22, -40) mm, rotated rx 180 ry 0 rz 0.01 deg; joints [29.421, -41.374, 97.382, -145.983, 61.451, 163.153]
  MoveC 3975 to (-322.59, 74.68, -40) mm, rotated rx -180 ry 0 rz 0.01 deg; joints [29.385, -41.532, 97.724, -146.077, 61.593, 163.288] to (-320.27, 71.92, -40) mm, rotated rx 180 ry 0 rz 0.01 deg; joints [29.339, -41.685, 98.055, -146.18, 61.726, 163.425]
  MoveC 3976 to (-318.09, 69.06, -40) mm, rotated rx -180 ry 0 rz 0.01 deg; joints [29.287, -41.834, 98.378, -146.289, 61.855, 163.562] to (-315.92, 66.18, -40) mm, rotated rx -180 ry 0 rz 0.01 deg; joints [29.233, -41.982, 98.699, -146.398, 61.982, 163.699]
  MoveL 3977 to (-295.35, 31.01, -40) mm, rotated rx 180 ry 0 rz 0.01 deg; joints [28.454, -43.519, 102.053, -147.749, 63.281, 165.205]
  MoveC 3978 to (-292.39, 25.06, -40) mm, rotated rx -180 ry 0 rz 0.01 deg; joints [28.309, -43.752, 102.565, -147.979, 63.477, 165.443] to (-290.18, 18.79, -40) mm, rotated rx -180 ry 0 rz 0.01 deg; joints [28.139, -43.961, 103.026, -148.228, 63.645, 165.675]
  MoveC 3979 to (-288.66, 12.32, -40) mm, rotated rx -180 ry 0 rz 0.01 deg; joints [27.949, -44.146, 103.436, -148.49, 63.786, 165.899] to (-287.73, 5.74, -40) mm, rotated rx 180 ry 0 rz 0.01 deg; joints [27.744, -44.308, 103.799, -148.762, 63.902, 166.114]
  MoveC 3980 to (-286.36, 3, -40) mm, rotated rx -180 ry 0 rz 0.01 deg; joints [27.675, -44.413, 104.03, -148.867, 63.992, 166.22] to (-283.5, 1.89, -40) mm, rotated rx 180 ry 0 rz 0.01 deg; joints [27.689, -44.543, 104.313, -148.892, 64.127, 166.302]
  MoveL 3981 to (-110.05, 1.89, -40) mm, rotated rx 180 ry 0 rz 0.01 deg; joints [31.13, -50.636, 117.653, -146.859, 71.083, 169.054]
  MoveC 3982 to (-107.13, 3.02, -40) mm, rotated rx 180 ry 0 rz 0.01 deg; joints [31.235, -50.709, 117.814, -146.767, 71.179, 169.068] to (-105.74, 5.81, -40) mm, rotated rx -180 ry 0 rz 0.01 deg; joints [31.368, -50.702, 117.792, -146.627, 71.195, 169.014]
  MoveC 3983 to (-104.79, 12.48, -40) mm, rotated rx -180 ry 0 rz 0.01 deg; joints [31.632, -50.608, 117.567, -146.33, 71.142, 168.847] to (-103.23, 19.03, -40) mm, rotated rx 180 ry 0 rz 0.01 deg; joints [31.904, -50.534, 117.388, -146.029, 71.115, 168.692]
  MoveC 3984 to (-100.98, 25.38, -40) mm, rotated rx 180 ry 0 rz 0.01 deg; joints [32.184, -50.486, 117.266, -145.727, 71.115, 168.551] to (-97.97, 31.41, -40) mm, rotated rx 180 ry 0 rz 0.01 deg; joints [32.469, -50.466, 117.209, -145.426, 71.148, 168.431]
  MoveL 3985 to (-77.06, 66.93, -40) mm, rotated rx 180 ry 0 rz 0.01 deg; joints [34.217, -50.424, 117.038, -143.604, 71.445, 167.757]
  MoveC 3986 to (-69, 75.98, -40) mm, rotated rx 180 ry 0 rz 0.01 deg; joints [34.728, -50.491, 117.167, -143.094, 71.616, 167.625] to (-59.77, 83.84, -40) mm, rotated rx -180 ry 0 rz 0.01 deg; joints [35.226, -50.615, 117.427, -142.611, 71.843, 167.546]
  MoveC 3987 to (-49.22, 89.9, -40) mm, rotated rx 180 ry 0 rz 0.01 deg; joints [35.698, -50.813, 117.855, -142.175, 72.138, 167.54] to (-37.57, 93.42, -40) mm, rotated rx 180 ry 0 rz 0.01 deg; joints [36.113, -51.093, 118.474, -141.818, 72.504, 167.626]
  MoveC 3988 to (-34.87, 93.86, -40) mm, rotated rx 180 ry 0 rz 0.01 deg; joints [36.197, -51.166, 118.636, -141.75, 72.593, 167.657] to (-32.14, 94.17, -40) mm, rotated rx -180 ry 0 rz 0.01 deg; joints [36.277, -51.242, 118.804, -141.687, 72.685, 167.692]
  MoveC 3989 to (-29.41, 94.39, -40) mm, rotated rx 180 ry 0 rz 0.01 deg; joints [36.355, -51.319, 118.977, -141.626, 72.778, 167.73] to (-26.68, 94.57, -40) mm, rotated rx -180 ry 0 rz 0.01 deg; joints [36.431, -51.398, 119.152, -141.567, 72.872, 167.769]
  MoveC 3990 to (-23.98, 95.82, -40) mm, rotated rx 180 ry 0 rz 0.01 deg; joints [36.544, -51.452, 119.271, -141.465, 72.949, 167.776] to (-22.88, 98.58, -40) mm, rotated rx 180 ry 0 rz 0.01 deg; joints [36.668, -51.426, 119.208, -141.331, 72.949, 167.713]
  MoveL 3991 to (-22.89, 302.2, -40) mm, rotated rx 180 ry 0 rz 0.01 deg; joints [43.112, -46.45, 107.89, -133.388, 70.16, 161.049]
  MoveC 3992 to (-24.02, 304.92, -40) mm, rotated rx 180 ry 0 rz 0.01 deg; joints [43.16, -46.34, 107.647, -133.306, 70.085, 160.93] to (-26.74, 306.05, -40) mm, rotated rx 180 ry 0 rz 0.01 deg; joints [43.119, -46.225, 107.398, -133.311, 69.978, 160.839]
  MoveL 3993 to (-110.8, 306.05, -40) mm, rotated rx -180 ry 0 rz 0.01 deg; joints [40.957, -43.536, 101.61, -134.597, 67.041, 159.259]
  MoveC 3994 to (-113.25, 304.96, -40) mm, rotated rx -180 ry 0 rz 0.01 deg; joints [40.866, -43.485, 101.502, -134.672, 66.967, 159.252] to (-114.06, 302.4, -40) mm, rotated rx -180 ry 0 rz 0.01 deg; joints [40.773, -43.529, 101.602, -134.782, 66.971, 159.332]
  MoveC 3995 to (-115.32, 282.6, -40) mm, rotated rx -180 ry 0 rz 0.01 deg; joints [40.174, -44.039, 102.725, -135.57, 67.184, 160.043] to (-123.28, 264.42, -40) mm, rotated rx 180 ry 0 rz 0.01 deg; joints [39.45, -44.266, 103.242, -136.387, 67.132, 160.554]
  MoveC 3996 to (-136.37, 249.66, -40) mm, rotated rx -180 ry 0 rz 0.01 deg; joints [38.7, -44.217, 103.16, -137.14, 66.844, 160.836] to (-152.98, 239.01, -40) mm, rotated rx 180 ry 0 rz 0.01 deg; joints [37.992, -43.928, 102.557, -137.771, 66.364, 160.899]
  MoveC 3997 to (-157.92, 237.08, -40) mm, rotated rx 180 ry 0 rz 0.01 deg; joints [37.819, -43.807, 102.301, -137.907, 66.203, 160.873] to (-163.06, 235.76, -40) mm, rotated rx 180 ry 0 rz 0.01 deg; joints [37.661, -43.662, 101.993, -138.021, 66.027, 160.821]
  MoveC 3998 to (-168.27, 234.82, -40) mm, rotated rx 180 ry 0 rz 0.01 deg; joints [37.513, -43.504, 101.656, -138.119, 65.842, 160.753] to (-173.51, 234.02, -40) mm, rotated rx -180 ry 0 rz 0.01 deg; joints [37.37, -43.34, 101.307, -138.211, 65.653, 160.68]
  MoveL 3999 to (-214.9, 233.67, -40) mm, rotated rx -180 ry 0 rz 0.01 deg; joints [36.436, -41.853, 98.134, -138.648, 64.055, 159.863]
  MoveC 4000 to (-240.66, 238.91, -40) mm, rotated rx -180 ry 0 rz 0.01 deg; joints [36.035, -40.745, 95.771, -138.651, 62.964, 159.127] to (-262.33, 253.8, -40) mm, rotated rx 180 ry 0 rz 0.01 deg; joints [36.009, -39.499, 93.11, -138.187, 61.895, 158.079]
  MoveC 4001 to (-274.91, 272.92, -40) mm, rotated rx -180 ry 0 rz 0.01 deg; joints [36.293, -38.46, 90.887, -137.46, 61.133, 157.031] to (-279.67, 295.3, -40) mm, rotated rx -180 ry 0 rz 0.01 deg; joints [36.822, -37.613, 89.071, -136.542, 60.646, 156.001]
  MoveC 4002 to (-278.42, 299.46, -40) mm, rotated rx 180 ry 0 rz 0.01 deg; joints [36.964, -37.54, 88.911, -136.362, 60.644, 155.859] to (-274.95, 302.08, -40) mm, rotated rx -180 ry 0 rz 0.01 deg; joints [37.109, -37.603, 89.039, -136.237, 60.754, 155.836]
  MoveC 4003 to (-271.41, 304.46, -40) mm, rotated rx -180 ry 0 rz 0.01 deg; joints [37.25, -37.675, 89.187, -136.121, 60.869, 155.824] to (-269.54, 308.3, -40) mm, rotated rx 180 ry 0 rz 0.01 deg; joints [37.396, -37.635, 89.098, -135.951, 60.897, 155.71]
  MoveC 4004 to (-269.25, 309.84, -40) mm, rotated rx -180 ry 0 rz 0.01 deg; joints [37.444, -37.6, 89.022, -135.886, 60.888, 155.652] to (-269, 311.39, -40) mm, rotated rx -180 ry 0 rz 0.01 deg; joints [37.492, -37.564, 88.943, -135.82, 60.879, 155.594]
  MoveC 4005 to (-269.73, 313.95, -40) mm, rotated rx 180 ry 0 rz 0.01 deg; joints [37.547, -37.456, 88.713, -135.715, 60.815, 155.468] to (-272.16, 315.06, -40) mm, rotated rx 180 ry 0 rz 0.01 deg; joints [37.527, -37.324, 88.434, -135.679, 60.701, 155.361]
  MoveL 4006 to (-375.8, 315.06, -40) mm, rotated rx 180 ry 0 rz 0.01 deg; joints [35.444, -32.798, 78.97, -135.731, 56.204, 152.471]
  MoveC 4007 to (-378.52, 313.93, -40) mm, rotated rx 180 ry 0 rz 0.01 deg; joints [35.361, -32.707, 78.781, -135.772, 56.095, 152.439] to (-379.65, 311.21, -40) mm, rotated rx -180 ry 0 rz 0.01 deg; joints [35.267, -32.743, 78.86, -135.892, 56.08, 152.532]
  MoveL 4008 to (-379.64, 88.7, -40) mm, rotated rx -180 ry 0 rz 0.01 deg; joints [28.827, -38.849, 92.008, -145.713, 58.9, 161.637]
  MoveC 4009 to (-378.57, 86.27, -40) mm, rotated rx 180 ry 0 rz 0.01 deg; joints [28.77, -38.951, 92.227, -145.815, 58.978, 161.747] to (-376.05, 85.43, -40) mm, rotated rx -180 ry 0 rz 0.01 deg; joints [28.787, -39.078, 92.497, -145.845, 59.102, 161.831]
  MoveC 4010 to (-355.32, 83.75, -40) mm, rotated rx 180 ry 0 rz 0.01 deg; joints [29.092, -39.992, 94.435, -145.848, 60.05, 162.325] to (-336.46, 75.01, -40) mm, rotated rx -180 ry 0 rz 0.01 deg; joints [29.148, -40.964, 96.514, -146.138, 60.986, 163.006]
  MoveC 4011 to (-332.63, 71.95, -40) mm, rotated rx 180 ry 0 rz 0.01 deg; joints [29.119, -41.186, 96.992, -146.248, 61.189, 163.185] to (-329.23, 68.43, -40) mm, rotated rx -180 ry 0 rz 0.01 deg; joints [29.067, -41.4, 97.454, -146.38, 61.379, 163.369]
  MoveC 4012 to (-326.13, 64.65, -40) mm, rotated rx -180 ry 0 rz 0.01 deg; joints [29.001, -41.606, 97.901, -146.523, 61.559, 163.555] to (-323.14, 60.78, -40) mm, rotated rx 180 ry 0 rz 0.01 deg; joints [28.93, -41.809, 98.339, -146.671, 61.735, 163.74]
  MoveL 4013 to (-303.16, 26.51, -40) mm, rotated rx 180 ry 0 rz 0.01 deg; joints [28.165, -43.305, 101.603, -147.996, 63, 165.208]
  MoveC 4014 to (-299.82, 19.5, -40) mm, rotated rx -180 ry 0 rz 0.01 deg; joints [27.991, -43.574, 102.194, -148.27, 63.226, 165.485] to (-297.6, 12.05, -40) mm, rotated rx 180 ry 0 rz 0.01 deg; joints [27.781, -43.806, 102.706, -148.569, 63.408, 165.753]
  MoveC 4015 to (-296.51, 4.37, -40) mm, rotated rx 180 ry 0 rz 0.01 deg; joints [27.542, -43.997, 103.131, -148.888, 63.544, 166.007] to (-296.5, -3.39, -40) mm, rotated rx -180 ry 0 rz 0.01 deg; joints [27.28, -44.145, 103.466, -149.217, 63.635, 166.242]
  MoveC 4016 to (-295.57, -6.02, -40) mm, rotated rx -180 ry 0 rz 0.01 deg; joints [27.207, -44.231, 103.655, -149.322, 63.705, 166.337] to (-293.01, -7.13, -40) mm, rotated rx 180 ry 0 rz 0.01 deg; joints [27.214, -44.35, 103.915, -149.35, 63.827, 166.413]
  MoveL 4017 to (-100.42, -7.13, -40) mm, rotated rx -180 ry 0 rz 0.01 deg; joints [31.012, -51.111, 118.735, -147.093, 71.567, 169.444]
  MoveC 4018 to (-97.92, -6.04, -40) mm, rotated rx 180 ry 0 rz 0.01 deg; joints [31.107, -51.171, 118.867, -147.007, 71.647, 169.453] to (-97.03, -3.46, -40) mm, rotated rx 180 ry 0 rz 0.01 deg; joints [31.222, -51.152, 118.82, -146.883, 71.647, 169.398]
  MoveC 4019 to (-95.71, 13.55, -40) mm, rotated rx -180 ry 0 rz 0.01 deg; joints [31.875, -50.879, 118.17, -146.142, 71.471, 168.959] to (-89.21, 29.32, -40) mm, rotated rx 180 ry 0 rz 0.01 deg; joints [32.595, -50.786, 117.926, -145.373, 71.503, 168.627]
  MoveL 4020 to (-72.01, 58.3, -40) mm, rotated rx 180 ry 0 rz 0.01 deg; joints [34.033, -50.757, 117.798, -143.877, 71.747, 168.085]
  MoveC 4021 to (-62, 70.84, -40) mm, rotated rx 180 ry 0 rz 0.01 deg; joints [34.718, -50.814, 117.899, -143.185, 71.94, 167.887] to (-48.72, 79.87, -40) mm, rotated rx -180 ry 0 rz 0.01 deg; joints [35.361, -51.037, 118.378, -142.577, 72.294, 167.84]
  MoveC 4022 to (-33.47, 84.79, -40) mm, rotated rx 180 ry 0 rz 0.01 deg; joints [35.916, -51.399, 119.176, -142.095, 72.769, 167.944] to (-17.46, 85.43, -40) mm, rotated rx 180 ry 0 rz 0.01 deg; joints [36.349, -51.865, 120.22, -141.764, 73.324, 168.183]
  MoveC 4023 to (-14.94, 86.27, -40) mm, rotated rx 180 ry 0 rz 0.01 deg; joints [36.444, -51.922, 120.347, -141.68, 73.4, 168.2] to (-13.87, 88.7, -40) mm, rotated rx 180 ry 0 rz 0.01 deg; joints [36.557, -51.903, 120.299, -141.56, 73.404, 168.147]
  MoveL 4024 to (-13.87, 311.22, -40) mm, rotated rx -180 ry 0 rz 0.01 deg; joints [43.614, -46.472, 107.923, -132.891, 70.343, 160.884]
  MoveC 4025 to (-15, 313.94, -40) mm, rotated rx -180 ry 0 rz 0.01 deg; joints [43.661, -46.361, 107.68, -132.81, 70.269, 160.764] to (-17.73, 315.07, -40) mm, rotated rx 180 ry 0 rz 0.01 deg; joints [43.619, -46.247, 107.431, -132.816, 70.162, 160.673]
  MoveL 4026 to (-121.35, 315.07, -40) mm, rotated rx 180 ry 0 rz 0.01 deg; joints [40.953, -42.922, 100.285, -134.384, 66.541, 158.708]
  MoveC 4027 to (-123.76, 313.97, -40) mm, rotated rx 180 ry 0 rz 0.01 deg; joints [40.864, -42.872, 100.18, -134.457, 66.468, 158.702] to (-124.49, 311.43, -40) mm, rotated rx 180 ry 0 rz 0.01 deg; joints [40.774, -42.92, 100.286, -134.565, 66.474, 158.784]
  MoveC 4028 to (-123.7, 306.39, -40) mm, rotated rx 180 ry 0 rz 0.01 deg; joints [40.651, -43.091, 100.658, -134.752, 66.569, 158.991] to (-122.83, 301.36, -40) mm, rotated rx -180 ry 0 rz 0.01 deg; joints [40.529, -43.263, 101.034, -134.937, 66.666, 159.199]
  MoveC 4029 to (-122.44, 296.24, -40) mm, rotated rx 180 ry 0 rz 0.01 deg; joints [40.392, -43.42, 101.378, -135.131, 66.747, 159.398] to (-123.1, 291.15, -40) mm, rotated rx 180 ry 0 rz 0.01 deg; joints [40.231, -43.54, 101.643, -135.338, 66.789, 159.576]
  MoveC 4030 to (-125.08, 283.79, -40) mm, rotated rx -180 ry 0 rz 0.01 deg; joints [39.97, -43.677, 101.948, -135.652, 66.813, 159.81] to (-127.5, 276.56, -40) mm, rotated rx -180 ry 0 rz 0.01 deg; joints [39.702, -43.794, 102.21, -135.967, 66.819, 160.03]
  MoveC 4031 to (-130.77, 269.64, -40) mm, rotated rx 180 ry 0 rz 0.01 deg; joints [39.422, -43.872, 102.387, -136.281, 66.789, 160.22] to (-135.21, 263.41, -40) mm, rotated rx -180 ry 0 rz 0.01 deg; joints [39.133, -43.889, 102.434, -136.583, 66.707, 160.361]
  MoveC 4032 to (-144.16, 254.86, -40) mm, rotated rx 180 ry 0 rz 0.01 deg; joints [38.669, -43.812, 102.283, -137.033, 66.487, 160.498] to (-154.64, 248.29, -40) mm, rotated rx 180 ry 0 rz 0.01 deg; joints [38.229, -43.625, 101.893, -137.422, 66.181, 160.533]
  MoveC 4033 to (-166.31, 244.1, -40) mm, rotated rx 180 ry 0 rz 0.01 deg; joints [37.834, -43.328, 101.265, -137.725, 65.796, 160.457] to (-178.62, 242.68, -40) mm, rotated rx -180 ry 0 rz 0.01 deg; joints [37.511, -42.931, 100.417, -137.92, 65.346, 160.265]
  MoveL 4034 to (-218.76, 242.95, -40) mm, rotated rx -180 ry 0 rz 0.01 deg; joints [36.625, -41.462, 97.286, -138.304, 63.784, 159.438]
  MoveC 4035 to (-230.67, 245.62, -40) mm, rotated rx 180 ry 0 rz 0.01 deg; joints [36.445, -40.943, 96.18, -138.296, 63.277, 159.087] to (-241.98, 250.2, -40) mm, rotated rx -180 ry 0 rz 0.01 deg; joints [36.336, -40.388, 94.996, -138.196, 62.766, 158.669]
  MoveC 4036 to (-252.17, 257.01, -40) mm, rotated rx -180 ry 0 rz 0.01 deg; joints [36.316, -39.807, 93.755, -137.987, 62.268, 158.182] to (-260.42, 266.07, -40) mm, rotated rx 180 ry 0 rz 0.01 deg; joints [36.402, -39.231, 92.523, -137.665, 61.816, 157.641]
  MoveC 4037 to (-265.15, 273.88, -40) mm, rotated rx 180 ry 0 rz 0.01 deg; joints [36.524, -38.822, 91.648, -137.368, 61.522, 157.222] to (-268.71, 282.29, -40) mm, rotated rx -180 ry 0 rz 0.01 deg; joints [36.687, -38.438, 90.826, -137.036, 61.267, 156.8]
  MoveC 4038 to (-270.75, 291.22, -40) mm, rotated rx -180 ry 0 rz 0.01 deg; joints [36.895, -38.095, 90.091, -136.673, 61.068, 156.387] to (-270.91, 300.37, -40) mm, rotated rx 180 ry 0 rz 0.01 deg; joints [37.147, -37.818, 89.493, -136.29, 60.943, 156.006]
  MoveC 4039 to (-270.57, 303.15, -40) mm, rotated rx 180 ry 0 rz 0.01 deg; joints [37.231, -37.748, 89.343, -136.172, 60.921, 155.899] to (-270.04, 305.9, -40) mm, rotated rx -180 ry 0 rz 0.01 deg; joints [37.318, -37.687, 89.21, -136.055, 60.907, 155.798]
  MoveC 4040 to (-269.78, 307.1, -40) mm, rotated rx -180 ry 0 rz 0.01 deg; joints [37.357, -37.662, 89.155, -136.003, 60.902, 155.754] to (-269.54, 308.3, -40) mm, rotated rx -180 ry 0 rz 0.01 deg; joints [37.396, -37.635, 89.098, -135.951, 60.897, 155.71]
  MoveC 4041 to (-267.62, 311.89, -40) mm, rotated rx -180 ry 0 rz 0.01 deg; joints [37.535, -37.604, 89.027, -135.792, 60.929, 155.607] to (-264.02, 313.77, -40) mm, rotated rx 180 ry 0 rz 0.01 deg; joints [37.663, -37.692, 89.21, -135.697, 61.053, 155.617]
  MoveC 4042 to (-260.36, 315.39, -40) mm, rotated rx 180 ry 0 rz 0.01 deg; joints [37.786, -37.79, 89.413, -135.612, 61.181, 155.639] to (-257.84, 318.48, -40) mm, rotated rx 180 ry 0 rz 0.01 deg; joints [37.925, -37.797, 89.423, -135.47, 61.244, 155.571]
  MoveC 4043 to (-257.36, 319.44, -40) mm, rotated rx -180 ry 0 rz 0.01 deg; joints [37.962, -37.787, 89.401, -135.428, 61.251, 155.542] to (-256.85, 320.39, -40) mm, rotated rx 180 ry 0 rz 0.01 deg; joints [37.998, -37.778, 89.381, -135.385, 61.259, 155.515]
  MoveC 4044 to (-256.89, 322.64, -40) mm, rotated rx 180 ry 0 rz 0.01 deg; joints [38.059, -37.708, 89.23, -135.292, 61.228, 155.42] to (-258.85, 323.76, -40) mm, rotated rx -180 ry 0 rz 0.01 deg; joints [38.048, -37.596, 88.992, -135.255, 61.134, 155.324]
  MoveL 4045 to (-384.49, 323.76, -40) mm, rotated rx -180 ry 0 rz 0.01 deg; joints [35.511, -32.097, 77.498, -135.296, 55.688, 151.78]
  MoveC 4046 to (-387.22, 322.63, -40) mm, rotated rx -180 ry 0 rz 0.01 deg; joints [35.429, -32.004, 77.306, -135.334, 55.577, 151.745] to (-388.34, 319.9, -40) mm, rotated rx 180 ry 0 rz 0.01 deg; joints [35.335, -32.041, 77.387, -135.454, 55.561, 151.839]
  MoveL 4047 to (-388.34, 76.98, -40) mm, rotated rx -180 ry 0 rz 0.01 deg; joints [28.316, -38.739, 91.796, -146.241, 58.644, 161.868]
  MoveC 4048 to (-387.22, 74.74, -40) mm, rotated rx 180 ry 0 rz 0.01 deg; joints [28.266, -38.838, 92.009, -146.335, 58.722, 161.972] to (-384.75, 74.31, -40) mm, rotated rx -180 ry 0 rz 0.01 deg; joints [28.293, -38.954, 92.255, -146.348, 58.839, 162.04]
  MoveC 4049 to (-382.04, 75.17, -40) mm, rotated rx 180 ry 0 rz 0.01 deg; joints [28.366, -39.051, 92.459, -146.304, 58.952, 162.067] to (-379.37, 76.13, -40) mm, rotated rx -180 ry 0 rz 0.01 deg; joints [28.441, -39.145, 92.655, -146.256, 59.062, 162.09]
  MoveC 4050 to (-376.63, 76.91, -40) mm, rotated rx -180 ry 0 rz 0.01 deg; joints [28.512, -39.245, 92.865, -146.214, 59.177, 162.12] to (-373.79, 77.21, -40) mm, rotated rx 180 ry 0 rz 0.01 deg; joints [28.569, -39.359, 93.106, -146.193, 59.301, 162.17]
  MoveC 4051 to (-364.63, 76.76, -40) mm, rotated rx -180 ry 0 rz 0.01 deg; joints [28.712, -39.757, 93.95, -146.183, 59.719, 162.377] to (-355.61, 75.06, -40) mm, rotated rx -180 ry 0 rz 0.01 deg; joints [28.814, -40.173, 94.834, -146.222, 60.141, 162.62]
  MoveC 4052 to (-347.03, 71.68, -40) mm, rotated rx -180 ry 0 rz 0.01 deg; joints [28.857, -40.603, 95.753, -146.33, 60.561, 162.909] to (-339.51, 66.34, -40) mm, rotated rx 180 ry 0 rz 0.01 deg; joints [28.819, -41.027, 96.665, -146.522, 60.955, 163.239]
  MoveC 4053 to (-336.51, 63.45, -40) mm, rotated rx 180 ry 0 rz 0.01 deg; joints [28.779, -41.212, 97.062, -146.63, 61.121, 163.394] to (-333.68, 60.41, -40) mm, rotated rx -180 ry 0 rz 0.01 deg; joints [28.731, -41.392, 97.452, -146.745, 61.281, 163.551]
  MoveC 4054 to (-331.09, 57.15, -40) mm, rotated rx 180 ry 0 rz 0.01 deg; joints [28.672, -41.566, 97.829, -146.87, 61.432, 163.709] to (-328.83, 53.64, -40) mm, rotated rx 180 ry 0 rz 0.01 deg; joints [28.599, -41.731, 98.187, -147.007, 61.572, 163.867]
  MoveL 4055 to (-309.56, 19.87, -40) mm, rotated rx -180 ry 0 rz 0.01 deg; joints [27.832, -43.187, 101.362, -148.323, 62.803, 165.303]
  MoveC 4056 to (-307.59, 14.62, -40) mm, rotated rx -180 ry 0 rz 0.01 deg; joints [27.692, -43.367, 101.759, -148.532, 62.95, 165.501] to (-305.92, 9.27, -40) mm, rotated rx -180 ry 0 rz 0.01 deg; joints [27.542, -43.537, 102.133, -148.748, 63.084, 165.695]
  MoveC 4057 to (-304.88, 3.75, -40) mm, rotated rx 180 ry 0 rz 0.01 deg; joints [27.375, -43.684, 102.461, -148.975, 63.193, 165.883] to (-304.78, -1.87, -40) mm, rotated rx -180 ry 0 rz 0.01 deg; joints [27.187, -43.795, 102.711, -149.214, 63.262, 166.056]
  MoveC 4058 to (-305.35, -7.16, -40) mm, rotated rx 180 ry 0 rz 0.01 deg; joints [26.999, -43.873, 102.888, -149.443, 63.298, 166.207] to (-306.35, -12.38, -40) mm, rotated rx 180 ry 0 rz 0.01 deg; joints [26.805, -43.933, 103.026, -149.672, 63.316, 166.347]
  MoveC 4059 to (-305.8, -14.76, -40) mm, rotated rx 180 ry 0 rz 0.01 deg; joints [26.734, -43.998, 103.172, -149.77, 63.367, 166.428] to (-303.6, -15.82, -40) mm, rotated rx 180 ry 0 rz 0.01 deg; joints [26.735, -44.104, 103.401, -149.799, 63.474, 166.497]
  MoveL 4060 to (-89.91, -15.82, -40) mm, rotated rx -180 ry 0 rz 0.01 deg; joints [30.923, -51.603, 119.859, -147.297, 72.08, 169.834]
  MoveC 4061 to (-87.71, -14.76, -40) mm, rotated rx 180 ry 0 rz 0.01 deg; joints [31.012, -51.653, 119.971, -147.216, 72.149, 169.839] to (-87.16, -12.38, -40) mm, rotated rx -180 ry 0 rz 0.01 deg; joints [31.113, -51.628, 119.907, -147.105, 72.138, 169.785]
  MoveC 4062 to (-88.16, -6.83, -40) mm, rotated rx -180 ry 0 rz 0.01 deg; joints [31.297, -51.496, 119.598, -146.885, 72.026, 169.623] to (-88.61, -1.21, -40) mm, rotated rx 180 ry 0 rz 0.01 deg; joints [31.494, -51.379, 119.323, -146.653, 71.934, 169.467]
  MoveC 4063 to (-88.46, 4.42, -40) mm, rotated rx 180 ry 0 rz 0.01 deg; joints [31.706, -51.28, 119.088, -146.411, 71.865, 169.318] to (-87.62, 10, -40) mm, rotated rx 180 ry 0 rz 0.01 deg; joints [31.929, -51.203, 118.902, -146.161, 71.821, 169.18]
  MoveC 4064 to (-86.9, 12.69, -40) mm, rotated rx -180 ry 0 rz 0.01 deg; joints [32.044, -51.175, 118.834, -146.036, 71.812, 169.118] to (-85.91, 15.3, -40) mm, rotated rx 180 ry 0 rz 0.01 deg; joints [32.162, -51.158, 118.789, -145.909, 71.814, 169.063]
  MoveC 4065 to (-84.79, 17.86, -40) mm, rotated rx 180 ry 0 rz 0.01 deg; joints [32.281, -51.145, 118.754, -145.783, 71.822, 169.011] to (-83.69, 20.42, -40) mm, rotated rx 180 ry 0 rz 0.01 deg; joints [32.4, -51.131, 118.717, -145.657, 71.828, 168.958]
  MoveL 4066 to (-64.49, 53.95, -40) mm, rotated rx 180 ry 0 rz 0.01 deg; joints [34.06, -51.079, 118.527, -143.928, 72.081, 168.328]
  MoveC 4067 to (-57.23, 63.41, -40) mm, rotated rx 180 ry 0 rz 0.01 deg; joints [34.572, -51.113, 118.583, -143.409, 72.215, 168.176] to (-47.78, 70.68, -40) mm, rotated rx 180 ry 0 rz 0.01 deg; joints [35.061, -51.256, 118.885, -142.939, 72.455, 168.12]
  MoveC 4068 to (-36.85, 75.39, -40) mm, rotated rx -180 ry 0 rz 0.01 deg; joints [35.5, -51.491, 119.403, -142.544, 72.78, 168.16] to (-25.13, 77.44, -40) mm, rotated rx 180 ry 0 rz 0.01 deg; joints [35.87, -51.802, 120.096, -142.24, 73.167, 168.29]
  MoveC 4069 to (-22.46, 77.48, -40) mm, rotated rx -180 ry 0 rz 0.01 deg; joints [35.94, -51.881, 120.273, -142.187, 73.261, 168.331] to (-19.8, 77.3, -40) mm, rotated rx -180 ry 0 rz 0.01 deg; joints [36.002, -51.964, 120.46, -142.143, 73.357, 168.379]
  MoveC 4070 to (-17.17, 76.89, -40) mm, rotated rx 180 ry 0 rz 0.01 deg; joints [36.055, -52.051, 120.656, -142.109, 73.455, 168.433] to (-14.58, 76.24, -40) mm, rotated rx -180 ry 0 rz 0.01 deg; joints [36.099, -52.141, 120.861, -142.085, 73.555, 168.493]
  MoveC 4071 to (-13.12, 75.77, -40) mm, rotated rx -180 ry 0 rz 0.01 deg; joints [36.12, -52.194, 120.981, -142.075, 73.613, 168.53] to (-11.67, 75.26, -40) mm, rotated rx 180 ry 0 rz 0.01 deg; joints [36.14, -52.247, 121.103, -142.068, 73.671, 168.568]
  MoveC 4072 to (-10.22, 74.75, -40) mm, rotated rx -180 ry 0 rz 0.01 deg; joints [36.159, -52.3, 121.224, -142.06, 73.729, 168.606] to (-8.75, 74.28, -40) mm, rotated rx -180 ry 0 rz 0.01 deg; joints [36.181, -52.353, 121.344, -142.051, 73.787, 168.643]
  MoveC 4073 to (-6.29, 74.71, -40) mm, rotated rx 180 ry 0 rz 0.01 deg; joints [36.26, -52.417, 121.487, -141.984, 73.867, 168.67] to (-5.17, 76.94, -40) mm, rotated rx 180 ry 0 rz 0.01 deg; joints [36.369, -52.404, 121.453, -141.87, 73.874, 168.625]
  MoveL 4074 to (-5.18, 319.91, -40) mm, rotated rx 180 ry 0 rz 0.01 deg; joints [44.099, -46.488, 107.946, -132.412, 70.517, 160.722]
  MoveC 4075 to (-6.31, 322.64, -40) mm, rotated rx -180 ry 0 rz 0.01 deg; joints [44.145, -46.378, 107.702, -132.331, 70.443, 160.602] to (-9.03, 323.77, -40) mm, rotated rx 180 ry 0 rz 0.01 deg; joints [44.102, -46.264, 107.454, -132.338, 70.338, 160.511]
  MoveL 4076 to (-134.62, 323.76, -40) mm, rotated rx -180 ry 0 rz 0.01 deg; joints [40.875, -42.216, 98.767, -134.207, 65.943, 158.105]
  MoveC 4077 to (-136.6, 322.65, -40) mm, rotated rx 180 ry 0 rz 0.01 deg; joints [40.796, -42.18, 98.692, -134.274, 65.884, 158.108] to (-136.67, 320.37, -40) mm, rotated rx 180 ry 0 rz 0.01 deg; joints [40.731, -42.244, 98.831, -134.363, 65.912, 158.195]
  MoveC 4078 to (-133.76, 313.95, -40) mm, rotated rx -180 ry 0 rz 0.01 deg; joints [40.62, -42.53, 99.45, -134.58, 66.102, 158.501] to (-131.65, 307.23, -40) mm, rotated rx -180 ry 0 rz 0.01 deg; joints [40.482, -42.796, 100.027, -134.818, 66.267, 158.801]
  MoveC 4079 to (-130.76, 300.2, -40) mm, rotated rx -180 ry 0 rz 0.01 deg; joints [40.304, -43.026, 100.528, -135.082, 66.391, 159.085] to (-131.56, 293.15, -40) mm, rotated rx -180 ry 0 rz 0.01 deg; joints [40.083, -43.196, 100.904, -135.367, 66.453, 159.334]
  MoveC 4080 to (-133.87, 284.89, -40) mm, rotated rx 180 ry 0 rz 0.01 deg; joints [39.79, -43.348, 101.241, -135.721, 66.476, 159.597] to (-136.85, 276.84, -40) mm, rotated rx -180 ry 0 rz 0.01 deg; joints [39.486, -43.468, 101.511, -136.074, 66.471, 159.837]
  MoveC 4081 to (-141.2, 269.36, -40) mm, rotated rx 180 ry 0 rz 0.01 deg; joints [39.164, -43.523, 101.64, -136.423, 66.408, 160.027] to (-147.36, 263.28, -40) mm, rotated rx -180 ry 0 rz 0.01 deg; joints [38.841, -43.475, 101.548, -136.739, 66.258, 160.129]
  MoveC 4082 to (-152.26, 259.79, -40) mm, rotated rx 180 ry 0 rz 0.01 deg; joints [38.623, -43.4, 101.392, -136.936, 66.12, 160.161] to (-157.34, 256.57, -40) mm, rotated rx -180 ry 0 rz 0.01 deg; joints [38.41, -43.31, 101.205, -137.124, 65.972, 160.179]
  MoveC 4083 to (-162.82, 254, -40) mm, rotated rx -180 ry 0 rz 0.01 deg; joints [38.207, -43.187, 100.947, -137.29, 65.799, 160.165] to (-168.69, 252.57, -40) mm, rotated rx -180 ry 0 rz 0.01 deg; joints [38.03, -43.019, 100.589, -137.414, 65.596, 160.101]
  MoveC 4084 to (-171.17, 252.21, -40) mm, rotated rx -180 ry 0 rz 0.01 deg; joints [37.962, -42.941, 100.424, -137.456, 65.507, 160.065] to (-173.63, 251.8, -40) mm, rotated rx -180 ry 0 rz 0.01 deg; joints [37.894, -42.864, 100.261, -137.499, 65.418, 160.031]
  MoveC 4085 to (-176.12, 251.49, -40) mm, rotated rx 180 ry 0 rz 0.01 deg; joints [37.827, -42.785, 100.091, -137.539, 65.328, 159.993] to (-178.62, 251.38, -40) mm, rotated rx 180 ry 0 rz 0.01 deg; joints [37.767, -42.698, 99.907, -137.571, 65.234, 159.947]
  MoveL 4086 to (-217.56, 251.56, -40) mm, rotated rx 180 ry 0 rz 0.01 deg; joints [36.903, -41.273, 96.872, -137.943, 63.72, 159.14]
  MoveC 4087 to (-227.76, 253.81, -40) mm, rotated rx 180 ry 0 rz 0.01 deg; joints [36.746, -40.83, 95.927, -137.937, 63.288, 158.838] to (-237.47, 257.64, -40) mm, rotated rx 180 ry 0 rz 0.01 deg; joints [36.648, -40.356, 94.917, -137.857, 62.852, 158.482]
  MoveC 4088 to (-246.24, 263.37, -40) mm, rotated rx -180 ry 0 rz 0.01 deg; joints [36.625, -39.859, 93.856, -137.684, 62.426, 158.067] to (-253.33, 271.1, -40) mm, rotated rx 180 ry 0 rz 0.01 deg; joints [36.695, -39.366, 92.802, -137.412, 62.04, 157.604]
  MoveC 4089 to (-257.8, 278.94, -40) mm, rotated rx 180 ry 0 rz 0.01 deg; joints [36.823, -38.967, 91.948, -137.115, 61.757, 157.19] to (-260.64, 287.5, -40) mm, rotated rx 180 ry 0 rz 0.01 deg; joints [37.004, -38.607, 91.176, -136.775, 61.531, 156.779]
  MoveC 4090 to (-261.84, 295.85, -40) mm, rotated rx 180 ry 0 rz 0.01 deg; joints [37.212, -38.315, 90.547, -136.434, 61.374, 156.411] to (-261.75, 304.29, -40) mm, rotated rx -180 ry 0 rz 0.01 deg; joints [37.449, -38.068, 90.015, -136.082, 61.268, 156.066]
  MoveC 4091 to (-260.44, 311.56, -40) mm, rotated rx 180 ry 0 rz 0.01 deg; joints [37.679, -37.903, 89.655, -135.772, 61.228, 155.796] to (-257.84, 318.48, -40) mm, rotated rx -180 ry 0 rz 0.01 deg; joints [37.925, -37.797, 89.423, -135.47, 61.244, 155.571]
  MoveC 4092 to (-255.3, 321.2, -40) mm, rotated rx 180 ry 0 rz 0.01 deg; joints [38.054, -37.815, 89.458, -135.344, 61.312, 155.519] to (-251.68, 322.01, -40) mm, rotated rx 180 ry 0 rz 0.01 deg; joints [38.154, -37.935, 89.709, -135.291, 61.448, 155.574]
  MoveC 4093 to (-248.06, 322.66, -40) mm, rotated rx -180 ry 0 rz 0.01 deg; joints [38.25, -38.058, 89.967, -135.245, 61.586, 155.634] to (-245.26, 325.03, -40) mm, rotated rx 180 ry 0 rz 0.01 deg; joints [38.376, -38.097, 90.045, -135.131, 61.669, 155.603]
  MoveC 4094 to (-243.76, 327.01, -40) mm, rotated rx -180 ry 0 rz 0.01 deg; joints [38.462, -38.095, 90.039, -135.041, 61.703, 155.556] to (-242.14, 328.88, -40) mm, rotated rx 180 ry 0 rz 0.01 deg; joints [38.549, -38.102, 90.051, -134.954, 61.744, 155.517]
  MoveC 4095 to (-241.8, 330.8, -40) mm, rotated rx -180 ry 0 rz 0.01 deg; joints [38.609, -38.057, 89.951, -134.873, 61.733, 155.445] to (-243.43, 331.87, -40) mm, rotated rx 180 ry 0 rz 0.01 deg; joints [38.602, -37.959, 89.745, -134.837, 61.653, 155.36]
  MoveL 4096 to (-392.6, 331.87, -40) mm, rotated rx 180 ry 0 rz 0.01 deg; joints [35.572, -31.429, 76.1, -134.875, 55.2, 151.116]
  MoveC 4097 to (-395.32, 330.74, -40) mm, rotated rx -180 ry 0 rz 0.01 deg; joints [35.491, -31.335, 75.904, -134.911, 55.088, 151.079] to (-396.45, 328.01, -40) mm, rotated rx 180 ry 0 rz 0.01 deg; joints [35.397, -31.373, 75.987, -135.032, 55.073, 151.175]
  MoveL 4098 to (-396.45, 62.47, -40) mm, rotated rx -180 ry 0 rz 0.01 deg; joints [27.73, -38.71, 91.759, -146.888, 58.443, 162.208]
  MoveC 4099 to (-395.33, 60.7, -40) mm, rotated rx 180 ry 0 rz 0.01 deg; joints [27.692, -38.797, 91.947, -146.962, 58.515, 162.295] to (-393.25, 60.93, -40) mm, rotated rx -180 ry 0 rz 0.01 deg; joints [27.734, -38.883, 92.127, -146.948, 58.608, 162.331]
  MoveC 4100 to (-391.49, 62.33, -40) mm, rotated rx 180 ry 0 rz 0.01 deg; joints [27.807, -38.928, 92.221, -146.883, 58.672, 162.319] to (-389.74, 63.74, -40) mm, rotated rx 180 ry 0 rz 0.01 deg; joints [27.88, -38.973, 92.313, -146.818, 58.736, 162.306]
  MoveC 4101 to (-387.86, 64.98, -40) mm, rotated rx -180 ry 0 rz 0.01 deg; joints [27.95, -39.027, 92.425, -146.76, 58.808, 162.302] to (-385.76, 65.84, -40) mm, rotated rx -180 ry 0 rz 0.01 deg; joints [28.012, -39.098, 92.575, -146.718, 58.893, 162.317]
  MoveC 4102 to (-380.54, 67.32, -40) mm, rotated rx -180 ry 0 rz 0.01 deg; joints [28.146, -39.29, 92.978, -146.64, 59.113, 162.375] to (-375.27, 68.67, -40) mm, rotated rx 180 ry 0 rz 0.01 deg; joints [28.277, -39.485, 93.388, -146.566, 59.336, 162.437]
  MoveC 4103 to (-369.86, 69.39, -40) mm, rotated rx 180 ry 0 rz 0.01 deg; joints [28.391, -39.699, 93.84, -146.518, 59.571, 162.525] to (-364.41, 68.93, -40) mm, rotated rx 180 ry 0 rz 0.01 deg; joints [28.47, -39.939, 94.349, -146.519, 59.821, 162.652]
  MoveC 4104 to (-356.99, 66.85, -40) mm, rotated rx -180 ry 0 rz 0.01 deg; joints [28.531, -40.295, 95.108, -146.58, 60.177, 162.874] to (-350.03, 63.55, -40) mm, rotated rx -180 ry 0 rz 0.01 deg; joints [28.546, -40.655, 95.879, -146.691, 60.525, 163.126]
  MoveC 4105 to (-343.78, 59.02, -40) mm, rotated rx 180 ry 0 rz 0.01 deg; joints [28.51, -41.01, 96.641, -146.856, 60.854, 163.401] to (-338.56, 53.34, -40) mm, rotated rx 180 ry 0 rz 0.01 deg; joints [28.419, -41.344, 97.362, -147.073, 61.151, 163.692]
  MoveL 4106 to (-317.72, 18.12, -40) mm, rotated rx -180 ry 0 rz 0.01 deg; joints [27.631, -42.9, 100.751, -148.451, 62.472, 165.213]
  MoveC 4107 to (-313.91, 8.74, -40) mm, rotated rx -180 ry 0 rz 0.01 deg; joints [27.385, -43.234, 101.485, -148.826, 62.746, 165.573] to (-312.77, -1.32, -40) mm, rotated rx 180 ry 0 rz 0.01 deg; joints [27.068, -43.473, 102.016, -149.246, 62.911, 165.903]
  MoveC 4108 to (-314.31, -11.32, -40) mm, rotated rx -180 ry 0 rz 0.01 deg; joints [26.705, -43.602, 102.313, -149.683, 62.96, 166.181] to (-318.33, -20.6, -40) mm, rotated rx 180 ry 0 rz 0.01 deg; joints [26.323, -43.617, 102.364, -150.106, 62.891, 166.394]
  MoveC 4109 to (-318.35, -22.82, -40) mm, rotated rx -180 ry 0 rz 0.01 deg; joints [26.248, -43.657, 102.454, -150.201, 62.915, 166.46] to (-316.43, -23.93, -40) mm, rotated rx 180 ry 0 rz 0.01 deg; joints [26.242, -43.752, 102.662, -150.236, 63.011, 166.526]
  MoveL 4110 to (-77.11, -23.93, -40) mm, rotated rx 180 ry 0 rz 0.01 deg; joints [30.906, -52.15, 121.112, -147.435, 72.671, 170.238]
  MoveC 4111 to (-75.17, -22.82, -40) mm, rotated rx 180 ry 0 rz 0.01 deg; joints [30.992, -52.191, 121.202, -147.355, 72.729, 170.239] to (-75.17, -20.58, -40) mm, rotated rx -180 ry 0 rz 0.01 deg; joints [31.077, -52.152, 121.108, -147.259, 72.699, 170.181]
  MoveC 4112 to (-78.71, -12.56, -40) mm, rotated rx 180 ry 0 rz 0.01 deg; joints [31.297, -51.897, 120.515, -146.974, 72.458, 169.918] to (-80.51, -3.98, -40) mm, rotated rx 180 ry 0 rz 0.01 deg; joints [31.576, -51.685, 120.017, -146.638, 72.275, 169.664]
  MoveC 4113 to (-80.31, 4.81, -40) mm, rotated rx -180 ry 0 rz 0.01 deg; joints [31.906, -51.53, 119.648, -146.261, 72.165, 169.433] to (-77.92, 13.26, -40) mm, rotated rx -180 ry 0 rz 0.01 deg; joints [32.272, -51.448, 119.443, -145.863, 72.14, 169.242]
  MoveL 4114 to (-57.46, 49.89, -40) mm, rotated rx -180 ry 0 rz 0.01 deg; joints [34.084, -51.377, 119.203, -143.974, 72.392, 168.554]
  MoveC 4115 to (-51.42, 57.75, -40) mm, rotated rx -180 ry 0 rz 0.01 deg; joints [34.513, -51.406, 119.25, -143.54, 72.503, 168.429] to (-43.54, 63.78, -40) mm, rotated rx -180 ry 0 rz 0.01 deg; joints [34.922, -51.525, 119.505, -143.147, 72.703, 168.384]
  MoveC 4116 to (-34.44, 67.67, -40) mm, rotated rx 180 ry 0 rz 0.01 deg; joints [35.288, -51.722, 119.938, -142.818, 72.974, 168.419] to (-24.69, 69.36, -40) mm, rotated rx 180 ry 0 rz 0.01 deg; joints [35.595, -51.981, 120.516, -142.564, 73.296, 168.527]
  MoveC 4117 to (-19.25, 69.22, -40) mm, rotated rx -180 ry 0 rz 0.01 deg; joints [35.729, -52.146, 120.888, -142.465, 73.49, 168.618] to (-13.91, 68.22, -40) mm, rotated rx -180 ry 0 rz 0.01 deg; joints [35.831, -52.325, 121.294, -142.402, 73.693, 168.732]
  MoveC 4118 to (-8.78, 66.44, -40) mm, rotated rx -180 ry 0 rz 0.01 deg; joints [35.9, -52.512, 121.722, -142.375, 73.898, 168.864] to (-3.94, 63.96, -40) mm, rotated rx -180 ry 0 rz 0.01 deg; joints [35.936, -52.704, 122.162, -142.381, 74.103, 169.011]
  MoveC 4119 to (-2.95, 63.28, -40) mm, rotated rx 180 ry 0 rz 0.01 deg; joints [35.938, -52.747, 122.26, -142.389, 74.147, 169.046] to (-2.04, 62.5, -40) mm, rotated rx 180 ry 0 rz 0.01 deg; joints [35.933, -52.789, 122.358, -142.403, 74.19, 169.083]
  MoveC 4120 to (-1.16, 61.69, -40) mm, rotated rx -180 ry 0 rz 0.01 deg; joints [35.927, -52.831, 122.455, -142.419, 74.232, 169.119] to (-0.25, 60.92, -40) mm, rotated rx -180 ry 0 rz 0.01 deg; joints [35.923, -52.874, 122.553, -142.432, 74.275, 169.156]
  MoveC 4121 to (1.83, 60.68, -40) mm, rotated rx -180 ry 0 rz 0.01 deg; joints [35.969, -52.939, 122.702, -142.4, 74.351, 169.195] to (2.94, 62.45, -40) mm, rotated rx -180 ry 0 rz 0.01 deg; joints [36.062, -52.936, 122.69, -142.305, 74.364, 169.164]
  MoveL 4122 to (2.93, 328.02, -40) mm, rotated rx 180 ry 0 rz 0.01 deg; joints [44.55, -46.5, 107.959, -131.964, 70.678, 160.569]
  MoveC 4123 to (1.8, 330.75, -40) mm, rotated rx -180 ry 0 rz 0.01 deg; joints [44.596, -46.389, 107.714, -131.884, 70.604, 160.448] to (-0.92, 331.88, -40) mm, rotated rx -180 ry 0 rz 0.01 deg; joints [44.552, -46.275, 107.467, -131.892, 70.499, 160.357]
  MoveL 4124 to (-150.04, 331.87, -40) mm, rotated rx -180 ry 0 rz 0.01 deg; joints [40.73, -41.44, 97.103, -134.063, 65.267, 157.468]
  MoveC 4125 to (-151.71, 330.77, -40) mm, rotated rx 180 ry 0 rz 0.01 deg; joints [40.66, -41.414, 97.049, -134.125, 65.219, 157.476] to (-151.34, 328.8, -40) mm, rotated rx 180 ry 0 rz 0.01 deg; joints [40.614, -41.485, 97.203, -134.198, 65.259, 157.561]
  MoveC 4126 to (-145.99, 322.14, -40) mm, rotated rx 180 ry 0 rz 0.01 deg; joints [40.556, -41.868, 98.029, -134.401, 65.544, 157.934] to (-142.01, 314.57, -40) mm, rotated rx 180 ry 0 rz 0.01 deg; joints [40.44, -42.227, 98.803, -134.653, 65.79, 158.309]
  MoveC 4127 to (-139.66, 306.35, -40) mm, rotated rx 180 ry 0 rz 0.01 deg; joints [40.264, -42.545, 99.493, -134.948, 65.984, 158.673] to (-139.13, 297.81, -40) mm, rotated rx -180 ry 0 rz 0.01 deg; joints [40.034, -42.805, 100.062, -135.277, 66.114, 159.008]
  MoveC 4128 to (-141.28, 286.32, -40) mm, rotated rx 180 ry 0 rz 0.01 deg; joints [39.654, -43.053, 100.609, -135.755, 66.184, 159.397] to (-146.49, 275.85, -40) mm, rotated rx -180 ry 0 rz 0.01 deg; joints [39.228, -43.163, 100.859, -136.231, 66.127, 159.683]
  MoveC 4129 to (-154.62, 267.38, -40) mm, rotated rx 180 ry 0 rz 0.01 deg; joints [38.79, -43.112, 100.765, -136.663, 65.934, 159.836] to (-165.04, 261.97, -40) mm, rotated rx -180 ry 0 rz 0.01 deg; joints [38.39, -42.894, 100.307, -136.997, 65.612, 159.828]
  MoveC 4130 to (-168.36, 260.99, -40) mm, rotated rx 180 ry 0 rz 0.01 deg; joints [38.284, -42.803, 100.115, -137.074, 65.499, 159.798] to (-171.73, 260.2, -40) mm, rotated rx 180 ry 0 rz 0.01 deg; joints [38.183, -42.706, 99.908, -137.143, 65.382, 159.76]
  MoveC 4131 to (-175.15, 259.67, -40) mm, rotated rx -180 ry 0 rz 0.01 deg; joints [38.089, -42.598, 99.68, -137.201, 65.258, 159.711] to (-178.62, 259.49, -40) mm, rotated rx 180 ry 0 rz 0.01 deg; joints [38.005, -42.479, 99.427, -137.246, 65.129, 159.647]
  MoveL 4132 to (-216.45, 259.6, -40) mm, rotated rx -180 ry 0 rz 0.01 deg; joints [37.161, -41.095, 96.481, -137.606, 63.661, 158.86]
  MoveC 4133 to (-225.04, 261.45, -40) mm, rotated rx 180 ry 0 rz 0.01 deg; joints [37.027, -40.722, 95.686, -137.603, 63.298, 158.605] to (-233.26, 264.57, -40) mm, rotated rx 180 ry 0 rz 0.01 deg; joints [36.938, -40.324, 94.839, -137.54, 62.931, 158.307]
  MoveC 4134 to (-240.72, 269.31, -40) mm, rotated rx -180 ry 0 rz 0.01 deg; joints [36.913, -39.906, 93.946, -137.401, 62.572, 157.959] to (-246.72, 275.79, -40) mm, rotated rx 180 ry 0 rz 0.01 deg; joints [36.97, -39.491, 93.058, -137.175, 62.247, 157.569]
  MoveC 4135 to (-250.39, 282.23, -40) mm, rotated rx -180 ry 0 rz 0.01 deg; joints [37.074, -39.163, 92.356, -136.933, 62.015, 157.229] to (-252.73, 289.26, -40) mm, rotated rx 180 ry 0 rz 0.01 deg; joints [37.222, -38.868, 91.723, -136.656, 61.83, 156.893]
  MoveC 4136 to (-253.81, 296.02, -40) mm, rotated rx -180 ry 0 rz 0.01 deg; joints [37.388, -38.628, 91.206, -136.382, 61.699, 156.594] to (-254.07, 302.87, -40) mm, rotated rx 180 ry 0 rz 0.01 deg; joints [37.574, -38.416, 90.749, -136.1, 61.6, 156.309]
  MoveC 4137 to (-253.09, 309.68, -40) mm, rotated rx 180 ry 0 rz 0.01 deg; joints [37.784, -38.251, 90.392, -135.811, 61.551, 156.052] to (-250.52, 316.06, -40) mm, rotated rx -180 ry 0 rz 0.01 deg; joints [38.015, -38.161, 90.193, -135.532, 61.572, 155.849]
  MoveC 4138 to (-248.65, 319.41, -40) mm, rotated rx 180 ry 0 rz 0.01 deg; joints [38.148, -38.134, 90.131, -135.383, 61.605, 155.755] to (-246.73, 322.73, -40) mm, rotated rx -180 ry 0 rz 0.01 deg; joints [38.281, -38.109, 90.073, -135.234, 61.639, 155.663]
  MoveC 4139 to (-246.02, 323.89, -40) mm, rotated rx -180 ry 0 rz 0.01 deg; joints [38.328, -38.102, 90.056, -135.182, 61.653, 155.632] to (-245.26, 325.03, -40) mm, rotated rx 180 ry 0 rz 0.01 deg; joints [38.376, -38.097, 90.045, -135.131, 61.669, 155.603]
  MoveL 4140 to (-245.08, 325.63, -39.83) mm, rotated rx 180 ry 0 rz 0.01 deg; joints [38.396, -38.093, 90.021, -135.102, 61.663, 155.576]
  MoveL 4141 to (-245.15, 326.09, -39.37) mm, rotated rx -180 ry 0 rz 0.01 deg; joints [38.407, -38.099, 89.987, -135.077, 61.64, 155.54]
  MoveL 4142 to (-245.22, 326.24, -38.73) mm, rotated rx -180 ry 0 rz 0.01 deg; joints [38.409, -38.121, 89.974, -135.061, 61.616, 155.511]
  Set speed (500.0 mm/s)
  MoveL 4143 to (-245.22, 326.24, 11) mm, rotated rx 180 ry 0 rz 0.01 deg; joints [38.388, -40.403, 90.121, -134.235, 60.106, 153.782]
  Set speed (500.0 mm/s)
  MoveL 4144 to (-398.5, 339.2, 11) mm, rotated rx -180 ry 0 rz 0.01 deg; joints [35.632, -33.026, 75.127, -133.489, 53.441, 148.81]
  Set speed (100.0 mm/s)
  MoveL 4145 to (-398.5, 339.2, -18.23) mm, rotated rx -180 ry 0 rz 0.01 deg; joints [35.645, -31.813, 75.06, -134.081, 54.241, 149.827]
  MoveL 4146 to (-398.51, 339.2, -18.37) mm, rotated rx -180 ry 0 rz 0.01 deg; joints [35.645, -31.806, 75.058, -134.083, 54.244, 149.831]
  MoveL 4147 to (-398.77, 339.19, -19.02) mm, rotated rx -180 ry 0 rz 0.01 deg; joints [35.64, -31.766, 75.029, -134.094, 54.249, 149.844]
  MoveL 4148 to (-399.34, 339.13, -19.43) mm, rotated rx -180 ry 0 rz 0.01 deg; joints [35.628, -31.723, 74.974, -134.101, 54.235, 149.841]
  MoveL 4149 to (-399.69, 339.08, -19.5) mm, rotated rx -180 ry 0 rz 0.01 deg; joints [35.62, -31.704, 74.941, -134.102, 54.221, 149.834]
  MoveL 4150 to (-399.72, 339.07, -19.5) mm, rotated rx -180 ry 0 rz 0.01 deg; joints [35.619, -31.703, 74.939, -134.102, 54.22, 149.833]
  MoveL 4151 to (-400.55, 338.85, -19.53) mm, rotated rx -180 ry 0 rz 0.01 deg; joints [35.597, -31.667, 74.869, -134.107, 54.184, 149.816]
  MoveL 4152 to (-400.6, 338.83, -19.53) mm, rotated rx -180 ry 0 rz 0.01 deg; joints [35.596, -31.665, 74.866, -134.107, 54.183, 149.816]
  MoveL 4153 to (-401.28, 338.49, -19.56) mm, rotated rx -180 ry 0 rz 0.01 deg; joints [35.574, -31.642, 74.82, -134.119, 54.156, 149.81]
  MoveL 4154 to (-401.4, 338.42, -19.56) mm, rotated rx -180 ry 0 rz 0.01 deg; joints [35.57, -31.638, 74.813, -134.121, 54.151, 149.809]
  MoveL 4155 to (-402.84, 337.05, -19.63) mm, rotated rx 180 ry 0 rz 0.01 deg; joints [35.507, -31.611, 74.764, -134.177, 54.103, 149.83]
  MoveL 4156 to (-402.87, 337.02, -19.63) mm, rotated rx -180 ry 0 rz 0.01 deg; joints [35.506, -31.611, 74.764, -134.178, 54.103, 149.831]
  MoveL 4157 to (-403.75, 334.43, -19.73) mm, rotated rx 180 ry 0 rz 0.01 deg; joints [35.421, -31.653, 74.863, -134.297, 54.098, 149.934]
  MoveL 4158 to (-403.78, 333.95, -19.75) mm, rotated rx -180 ry 0 rz 0.01 deg; joints [35.408, -31.668, 74.896, -134.32, 54.103, 149.958]
  MoveL 4159 to (-403.79, 333.65, -19.76) mm, rotated rx -180 ry 0 rz 0.01 deg; joints [35.4, -31.678, 74.916, -134.334, 54.107, 149.973]
  MoveL 4160 to (-403.79, 333.05, -19.78) mm, rotated rx -180 ry 0 rz 0.01 deg; joints [35.384, -31.698, 74.961, -134.363, 54.115, 150.004]
  MoveL 4161 to (-401.25, 328.08, -19.98) mm, rotated rx -180 ry 0 rz 0.01 deg; joints [35.3, -31.99, 75.584, -134.622, 54.305, 150.349]
  MoveL 4162 to (-395.74, 327.2, -20.18) mm, rotated rx -180 ry 0 rz 0.01 deg; joints [35.381, -32.285, 76.21, -134.705, 54.578, 150.587]
  MoveL 4163 to (-391.79, 331.15, -20.39) mm, rotated rx -180 ry 0 rz 0.01 deg; joints [35.56, -32.335, 76.325, -134.549, 54.715, 150.532]
  MoveL 4164 to (-392.66, 336.66, -20.59) mm, rotated rx 180 ry 0 rz 0.01 deg; joints [35.689, -32.092, 75.834, -134.288, 54.609, 150.236]
  MoveL 4165 to (-397.64, 339.2, -20.79) mm, rotated rx -180 ry 0 rz 0.01 deg; joints [35.662, -31.748, 75.138, -134.137, 54.35, 149.943]
  MoveL 4166 to (-398.51, 339.2, -20.82) mm, rotated rx -180 ry 0 rz 0.01 deg; joints [35.646, -31.703, 75.049, -134.131, 54.31, 149.914]
  MoveL 4167 to (-399.34, 339.13, -20.85) mm, rotated rx -180 ry 0 rz 0.01 deg; joints [35.628, -31.662, 74.968, -134.128, 54.273, 149.889]
  MoveL 4168 to (-399.69, 339.08, -20.86) mm, rotated rx 180 ry 0 rz 0.01 deg; joints [35.62, -31.646, 74.936, -134.128, 54.258, 149.88]
  MoveL 4169 to (-400.55, 338.85, -20.89) mm, rotated rx -180 ry 0 rz 0.01 deg; joints [35.598, -31.61, 74.864, -134.133, 54.221, 149.862]
  MoveL 4170 to (-400.6, 338.83, -20.9) mm, rotated rx -180 ry 0 rz 0.01 deg; joints [35.597, -31.608, 74.86, -134.134, 54.219, 149.862]
  MoveL 4171 to (-401.28, 338.49, -20.92) mm, rotated rx -180 ry 0 rz 0.01 deg; joints [35.575, -31.584, 74.814, -134.145, 54.192, 149.856]
  MoveL 4172 to (-401.4, 338.42, -20.93) mm, rotated rx -180 ry 0 rz 0.01 deg; joints [35.571, -31.581, 74.807, -134.148, 54.188, 149.855]
  MoveL 4173 to (-402.84, 337.05, -21) mm, rotated rx -180 ry 0 rz 0.01 deg; joints [35.508, -31.553, 74.759, -134.203, 54.14, 149.876]
  MoveL 4174 to (-402.87, 337.02, -21) mm, rotated rx -180 ry 0 rz 0.01 deg; joints [35.506, -31.553, 74.759, -134.205, 54.14, 149.877]
  MoveL 4175 to (-403.75, 334.43, -21.1) mm, rotated rx -180 ry 0 rz 0.01 deg; joints [35.422, -31.596, 74.858, -134.323, 54.135, 149.98]
  MoveL 4176 to (-403.78, 333.95, -21.11) mm, rotated rx -180 ry 0 rz 0.01 deg; joints [35.408, -31.611, 74.89, -134.346, 54.14, 150.004]
  MoveL 4177 to (-403.79, 333.65, -21.12) mm, rotated rx 180 ry 0 rz 0.01 deg; joints [35.4, -31.62, 74.911, -134.36, 54.144, 150.019]
  MoveL 4178 to (-403.79, 333.05, -21.14) mm, rotated rx -180 ry 0 rz 0.01 deg; joints [35.384, -31.64, 74.955, -134.39, 54.152, 150.05]
  MoveL 4179 to (-401.25, 328.08, -21.35) mm, rotated rx -180 ry 0 rz 0.01 deg; joints [35.301, -31.932, 75.579, -134.648, 54.342, 150.394]
  MoveL 4180 to (-395.74, 327.2, -21.55) mm, rotated rx 180 ry 0 rz 0.01 deg; joints [35.381, -32.227, 76.205, -134.731, 54.616, 150.633]
  MoveL 4181 to (-391.79, 331.15, -21.75) mm, rotated rx 180 ry 0 rz 0.01 deg; joints [35.561, -32.277, 76.319, -134.575, 54.753, 150.578]
  MoveL 4182 to (-392.66, 336.66, -21.95) mm, rotated rx -180 ry 0 rz 0.01 deg; joints [35.69, -32.034, 75.829, -134.314, 54.646, 150.281]
  MoveL 4183 to (-397.64, 339.2, -22.16) mm, rotated rx -180 ry 0 rz 0.01 deg; joints [35.663, -31.69, 75.133, -134.163, 54.387, 149.989]
  MoveL 4184 to (-398.51, 339.2, -22.19) mm, rotated rx -180 ry 0 rz 0.01 deg; joints [35.646, -31.645, 75.044, -134.157, 54.347, 149.96]
  MoveL 4185 to (-399.34, 339.13, -22.22) mm, rotated rx 180 ry 0 rz 0.01 deg; joints [35.629, -31.605, 74.963, -134.155, 54.31, 149.935]
  MoveL 4186 to (-399.69, 339.08, -22.23) mm, rotated rx -180 ry 0 rz 0.01 deg; joints [35.621, -31.588, 74.93, -134.155, 54.294, 149.926]
  MoveL 4187 to (-400.55, 338.85, -22.26) mm, rotated rx 180 ry 0 rz 0.01 deg; joints [35.599, -31.552, 74.858, -134.16, 54.258, 149.908]
  MoveL 4188 to (-400.6, 338.83, -22.26) mm, rotated rx -180 ry 0 rz 0.01 deg; joints [35.597, -31.55, 74.855, -134.16, 54.256, 149.908]
  MoveL 4189 to (-401.28, 338.49, -22.29) mm, rotated rx -180 ry 0 rz 0.01 deg; joints [35.576, -31.527, 74.809, -134.172, 54.229, 149.902]
  MoveL 4190 to (-401.4, 338.42, -22.29) mm, rotated rx -180 ry 0 rz 0.01 deg; joints [35.571, -31.523, 74.802, -134.174, 54.225, 149.901]
  MoveL 4191 to (-402.84, 337.05, -22.36) mm, rotated rx -180 ry 0 rz 0.01 deg; joints [35.508, -31.496, 74.754, -134.23, 54.177, 149.922]
  MoveL 4192 to (-402.87, 337.02, -22.36) mm, rotated rx -180 ry 0 rz 0.01 deg; joints [35.507, -31.496, 74.754, -134.231, 54.176, 149.923]
  MoveL 4193 to (-403.75, 334.43, -22.46) mm, rotated rx -180 ry 0 rz 0.01 deg; joints [35.422, -31.538, 74.852, -134.35, 54.171, 150.026]
  MoveL 4194 to (-403.78, 333.95, -22.48) mm, rotated rx -180 ry 0 rz 0.01 deg; joints [35.409, -31.553, 74.885, -134.373, 54.177, 150.05]
  MoveL 4195 to (-403.79, 333.65, -22.49) mm, rotated rx -180 ry 0 rz 0.01 deg; joints [35.401, -31.562, 74.906, -134.387, 54.181, 150.065]
  MoveL 4196 to (-403.79, 333.05, -22.51) mm, rotated rx -180 ry 0 rz 0.01 deg; joints [35.385, -31.583, 74.95, -134.416, 54.189, 150.096]
  MoveL 4197 to (-401.25, 328.08, -22.71) mm, rotated rx 180 ry 0 rz 0.01 deg; joints [35.301, -31.874, 75.574, -134.675, 54.379, 150.44]
  MoveL 4198 to (-395.74, 327.2, -22.91) mm, rotated rx 180 ry 0 rz 0.01 deg; joints [35.382, -32.169, 76.199, -134.757, 54.653, 150.678]
  MoveL 4199 to (-391.79, 331.15, -23.12) mm, rotated rx 180 ry 0 rz 0.01 deg; joints [35.561, -32.219, 76.314, -134.601, 54.79, 150.624]
  MoveL 4200 to (-392.66, 336.66, -23.32) mm, rotated rx -180 ry 0 rz 0.01 deg; joints [35.691, -31.976, 75.823, -134.34, 54.683, 150.327]
  MoveL 4201 to (-397.64, 339.2, -23.52) mm, rotated rx 180 ry 0 rz 0.01 deg; joints [35.663, -31.632, 75.128, -134.189, 54.423, 150.035]
  MoveL 4202 to (-398.51, 339.2, -23.55) mm, rotated rx 180 ry 0 rz 0.01 deg; joints [35.647, -31.587, 75.038, -134.183, 54.384, 150.006]
  MoveL 4203 to (-399.34, 339.13, -23.58) mm, rotated rx 180 ry 0 rz 0.01 deg; joints [35.63, -31.547, 74.957, -134.181, 54.347, 149.981]
  MoveL 4204 to (-399.69, 339.08, -23.59) mm, rotated rx 180 ry 0 rz 0.01 deg; joints [35.621, -31.531, 74.925, -134.181, 54.331, 149.972]
  MoveL 4205 to (-400.55, 338.85, -23.62) mm, rotated rx -180 ry 0 rz 0.01 deg; joints [35.599, -31.494, 74.853, -134.186, 54.295, 149.954]
  MoveL 4206 to (-400.6, 338.83, -23.63) mm, rotated rx -180 ry 0 rz 0.01 deg; joints [35.598, -31.493, 74.85, -134.187, 54.293, 149.953]
  MoveL 4207 to (-401.28, 338.49, -23.65) mm, rotated rx -180 ry 0 rz 0.01 deg; joints [35.576, -31.469, 74.804, -134.198, 54.266, 149.947]
  MoveL 4208 to (-401.4, 338.42, -23.66) mm, rotated rx 180 ry 0 rz 0.01 deg; joints [35.572, -31.465, 74.796, -134.201, 54.261, 149.947]
  MoveL 4209 to (-402.84, 337.05, -23.73) mm, rotated rx 180 ry 0 rz 0.01 deg; joints [35.509, -31.438, 74.748, -134.256, 54.214, 149.968]
  MoveL 4210 to (-402.87, 337.02, -23.73) mm, rotated rx -180 ry 0 rz 0.01 deg; joints [35.507, -31.438, 74.748, -134.258, 54.213, 149.969]
  MoveL 4211 to (-403.75, 334.43, -23.83) mm, rotated rx -180 ry 0 rz 0.01 deg; joints [35.423, -31.48, 74.847, -134.376, 54.208, 150.071]
  MoveL 4212 to (-403.78, 333.95, -23.84) mm, rotated rx -180 ry 0 rz 0.01 deg; joints [35.409, -31.495, 74.88, -134.399, 54.214, 150.095]
  MoveL 4213 to (-403.79, 333.65, -23.85) mm, rotated rx 180 ry 0 rz 0.01 deg; joints [35.402, -31.505, 74.9, -134.413, 54.218, 150.11]
  MoveL 4214 to (-403.79, 333.05, -23.87) mm, rotated rx -180 ry 0 rz 0.01 deg; joints [35.386, -31.525, 74.944, -134.442, 54.226, 150.141]
  MoveL 4215 to (-401.25, 328.08, -24.08) mm, rotated rx -180 ry 0 rz 0.01 deg; joints [35.302, -31.816, 75.568, -134.701, 54.416, 150.485]
  MoveL 4216 to (-395.74, 327.2, -24.28) mm, rotated rx -180 ry 0 rz 0.01 deg; joints [35.382, -32.111, 76.194, -134.783, 54.69, 150.724]
  MoveL 4217 to (-391.79, 331.15, -24.48) mm, rotated rx -180 ry 0 rz 0.01 deg; joints [35.562, -32.161, 76.308, -134.627, 54.827, 150.669]
  MoveL 4218 to (-392.66, 336.66, -24.68) mm, rotated rx -180 ry 0 rz 0.01 deg; joints [35.691, -31.918, 75.818, -134.366, 54.72, 150.373]
  MoveL 4219 to (-397.64, 339.2, -24.89) mm, rotated rx 180 ry 0 rz 0.01 deg; joints [35.664, -31.574, 75.122, -134.215, 54.46, 150.081]
  MoveL 4220 to (-398.51, 339.2, -24.92) mm, rotated rx -180 ry 0 rz 0.01 deg; joints [35.647, -31.53, 75.033, -134.21, 54.42, 150.051]
